	CONST robtarget Target_3690:=[[1119.7,-188.1,-317.9],[-0.081770019911019,-0.37959293775452,0.909310655383545,0.149589429628541],[-1,0,0,1],[9E+09,9E+09,9E+09,9E+09,9E+09,9E+09]];
	CONST robtarget Target_3700:=[[1124.4,-187.9,-319.1],[-0.0822084087134797,-0.376924329069528,0.910420076965927,0.149348957644967],[-1,0,0,1],[9E+09,9E+09,9E+09,9E+09,9E+09,9E+09]];
	CONST robtarget Target_3710:=[[1129.1,-187.6,-320.4],[-0.082652076021253,-0.374348316571166,0.911487931806646,0.14906952197064],[-1,0,0,1],[9E+09,9E+09,9E+09,9E+09,9E+09,9E+09]];
	CONST robtarget Target_3720:=[[1133.8,-187.2,-321.6],[-0.0830604381900551,-0.371848073764742,0.912510779106895,0.148842371853092],[-1,0,0,1],[9E+09,9E+09,9E+09,9E+09,9E+09,9E+09]];
	CONST robtarget Target_3730:=[[1138.6,-187,-322.9],[-0.0834905201851688,-0.369207677745856,0.913582291116862,0.148601551440044],[-1,0,0,1],[9E+09,9E+09,9E+09,9E+09,9E+09,9E+09]];
	CONST robtarget Target_3740:=[[1143.3,-186.7,-324.1],[-0.0839164170034894,-0.366716795237724,0.914590588848913,0.148326942383598],[-1,0,0,1],[9E+09,9E+09,9E+09,9E+09,9E+09,9E+09]];
	CONST robtarget Target_3750:=[[1148,-186.4,-325.4],[-0.0843167371331287,-0.364245178298671,0.915577742852347,0.14809974584311],[-1,0,0,1],[9E+09,9E+09,9E+09,9E+09,9E+09,9E+09]];
	CONST robtarget Target_3760:=[[1152.7,-186.1,-326.6],[-0.0847116064048817,-0.361800877254619,0.916546386353804,0.147874239203031],[-1,0,0,1],[9E+09,9E+09,9E+09,9E+09,9E+09,9E+09]];
	CONST robtarget Target_3770:=[[1157.5,-185.8,-327.9],[-0.0851099118523378,-0.359328899108832,0.917518335176831,0.147645351379778],[-1,0,0,1],[9E+09,9E+09,9E+09,9E+09,9E+09,9E+09]];
	CONST robtarget Target_3780:=[[1157.5,-180.9,-326.9],[-0.085634841189232,-0.362538132200784,0.916590329863401,0.145240985523245],[-1,0,0,1],[9E+09,9E+09,9E+09,9E+09,9E+09,9E+09]];
	CONST robtarget Target_3790:=[[1157.5,-176,-325.8],[-0.0861677390911265,-0.365697677609429,0.915653113093589,0.142897536063477],[-1,0,0,1],[9E+09,9E+09,9E+09,9E+09,9E+09,9E+09]];
	CONST robtarget Target_3800:=[[1157.5,-171.1,-324.9],[-0.0867279055318608,-0.368816467199481,0.914709329423617,0.140568583225226],[-1,0,0,1],[9E+09,9E+09,9E+09,9E+09,9E+09,9E+09]];
	CONST robtarget Target_3810:=[[1157.5,-166.2,-323.9],[-0.0873065476042629,-0.371898546178329,0.913760797007033,0.138239805949448],[-1,0,0,1],[9E+09,9E+09,9E+09,9E+09,9E+09,9E+09]];
	CONST robtarget Target_3820:=[[1157.5,-161.3,-323],[-0.087923551535875,-0.374952346833089,0.912809279452066,0.135865396756779],[-1,0,0,1],[9E+09,9E+09,9E+09,9E+09,9E+09,9E+09]];
	CONST robtarget Target_3830:=[[1157.5,-156.5,-322.1],[-0.0885457305098963,-0.377910274200135,0.911873087948939,0.133532579309003],[-1,0,0,1],[9E+09,9E+09,9E+09,9E+09,9E+09,9E+09]];
	CONST robtarget Target_3840:=[[1157.5,-151.6,-321.2],[-0.0891774776768113,-0.380884851594658,0.910911188916038,0.131205614241488],[-1,0,0,1],[9E+09,9E+09,9E+09,9E+09,9E+09,9E+09]];
	CONST robtarget Target_3850:=[[1157.5,-146.7,-320.4],[-0.0898350121694737,-0.383820989667297,0.909943857926704,0.128892567282967],[-1,0,0,1],[9E+09,9E+09,9E+09,9E+09,9E+09,9E+09]];
	CONST robtarget Target_3860:=[[1157.5,-141.8,-319.6],[-0.090538948270863,-0.386727190520538,0.908972312148108,0.126546887382584],[-1,0,0,1],[9E+09,9E+09,9E+09,9E+09,9E+09,9E+09]];
	CONST robtarget Target_3870:=[[1157.5,-136.9,-318.8],[-0.0912298198832608,-0.389593997110689,0.907997372118494,0.124235299352858],[-1,0,0,1],[9E+09,9E+09,9E+09,9E+09,9E+09,9E+09]];
	CONST robtarget Target_3880:=[[1157.5,-132,-318.1],[-0.091945722049869,-0.392423813800334,0.907017578768495,0.121937059026639],[-1,0,0,1],[9E+09,9E+09,9E+09,9E+09,9E+09,9E+09]];
	CONST robtarget Target_3890:=[[1157.5,-127.1,-317.4],[-0.09267744685106,-0.395219958040731,0.906034447792381,0.119639688335463],[-1,0,0,1],[9E+09,9E+09,9E+09,9E+09,9E+09,9E+09]];
	CONST robtarget Target_3900:=[[1157.5,-122.2,-316.7],[-0.0934459398585867,-0.397990450533941,0.90504850520611,0.117297318093474],[-1,0,0,1],[9E+09,9E+09,9E+09,9E+09,9E+09,9E+09]];
	CONST robtarget Target_3910:=[[1157.5,-117.3,-316],[-0.0942176050684812,-0.400717638074019,0.904057659766507,0.115013761129028],[-1,0,0,1],[9E+09,9E+09,9E+09,9E+09,9E+09,9E+09]];
	CONST robtarget Target_3920:=[[1157.5,-112.4,-315.4],[-0.0950042127207623,-0.403412314824983,0.903063888470925,0.112731172053829],[-1,0,0,1],[9E+09,9E+09,9E+09,9E+09,9E+09,9E+09]];
	CONST robtarget Target_3930:=[[1157.5,-107.6,-314.7],[-0.0958203709921909,-0.406026876380138,0.902086535754033,0.11045593769099],[-1,0,0,1],[9E+09,9E+09,9E+09,9E+09,9E+09,9E+09]];
	CONST robtarget Target_3940:=[[1157.5,-102.7,-314.2],[-0.0966575256864694,-0.408665629753412,0.901086967457954,0.108129565169957],[-1,0,0,1],[9E+09,9E+09,9E+09,9E+09,9E+09,9E+09]];
	CONST robtarget Target_3950:=[[1157.5,-97.8,-313.6],[-0.0974965183603951,-0.411263091531744,0.900083594760464,0.10586132860698],[-1,0,0,1],[9E+09,9E+09,9E+09,9E+09,9E+09,9E+09]];
	CONST robtarget Target_3960:=[[1157.5,-92.9,-313.1],[-0.0983493052491232,-0.413829493044003,0.899077740529287,0.103594311275819],[-1,0,0,1],[9E+09,9E+09,9E+09,9E+09,9E+09,9E+09]];
	CONST robtarget Target_3970:=[[1157.5,-88,-312.6],[-0.0992252665873052,-0.416363081924884,0.898068247921142,0.101338800844204],[-1,0,0,1],[9E+09,9E+09,9E+09,9E+09,9E+09,9E+09]];
	CONST robtarget Target_3980:=[[1157.5,-83.1,-312.1],[-0.100136755641848,-0.418873626645508,0.897055691069865,0.0990383874542113],[-1,0,0,1],[9E+09,9E+09,9E+09,9E+09,9E+09,9E+09]];
	CONST robtarget Target_3990:=[[1157.5,-78.2,-311.6],[-0.101039180167052,-0.421346926627475,0.896041552749548,0.0967852635421828],[-1,0,0,1],[9E+09,9E+09,9E+09,9E+09,9E+09,9E+09]];
	CONST robtarget Target_4000:=[[1157.5,-73.3,-311.2],[-0.101954320538193,-0.423790577515119,0.89502528752291,0.0945335793648495],[-1,0,0,1],[9E+09,9E+09,9E+09,9E+09,9E+09,9E+09]];
	CONST robtarget Target_4010:=[[1157.5,-68.5,-310.8],[-0.102896186994666,-0.42616193510684,0.894025342835322,0.0922879522805532],[-1,0,0,1],[9E+09,9E+09,9E+09,9E+09,9E+09,9E+09]];
	CONST robtarget Target_4020:=[[1157.5,-63.6,-310.5],[-0.103868543102495,-0.428553079264927,0.893002320186698,0.090002445230613],[-1,0,0,1],[9E+09,9E+09,9E+09,9E+09,9E+09,9E+09]];
	CONST robtarget Target_4030:=[[1157.5,-58.7,-310.1],[-0.104830406221372,-0.430908588307866,0.891978581406433,0.0877643707101632],[-1,0,0,1],[9E+09,9E+09,9E+09,9E+09,9E+09,9E+09]];
	CONST robtarget Target_4040:=[[1157.5,-53.8,-309.8],[-0.105814334622865,-0.433234255109494,0.890951696495378,0.0855364325889902],[-1,0,0,1],[9E+09,9E+09,9E+09,9E+09,9E+09,9E+09]];
	CONST robtarget Target_4050:=[[1157.5,-48.9,-309.5],[-0.106809880606017,-0.435532061690535,0.889922999304026,0.0833098310780098],[-1,0,0,1],[9E+09,9E+09,9E+09,9E+09,9E+09,9E+09]];
	CONST robtarget Target_4060:=[[1157.5,-44,-309.3],[-0.107839723601408,-0.437809013192539,0.888890636361769,0.0810388707307653],[-1,0,0,1],[9E+09,9E+09,9E+09,9E+09,9E+09,9E+09]];
	CONST robtarget Target_4070:=[[1157.5,-39.1,-309.1],[-0.10886840289795,-0.4400505689674,0.887857005220818,0.0788232572419922],[-1,0,0,1],[9E+09,9E+09,9E+09,9E+09,9E+09,9E+09]];
	CONST robtarget Target_4080:=[[1157.5,-34.2,-308.8],[-0.109897288481995,-0.442266525786448,0.886823054715504,0.0766014084606349],[-1,0,0,1],[9E+09,9E+09,9E+09,9E+09,9E+09,9E+09]];
	CONST robtarget Target_4090:=[[1157.5,-29.3,-308.7],[-0.110947538224501,-0.444454570827599,0.885786132357125,0.0743888832836221],[-1,0,0,1],[9E+09,9E+09,9E+09,9E+09,9E+09,9E+09]];
	CONST robtarget Target_4100:=[[1157.5,-24.4,-308.5],[-0.112042503144085,-0.44662162946331,0.884743749945618,0.0721394102894673],[-1,0,0,1],[9E+09,9E+09,9E+09,9E+09,9E+09,9E+09]];
	CONST robtarget Target_4110:=[[1157.5,-19.6,-308.4],[-0.113116403345818,-0.448720948594571,0.883722022425974,0.0699255079769918],[-1,0,0,1],[9E+09,9E+09,9E+09,9E+09,9E+09,9E+09]];
	CONST robtarget Target_4120:=[[1157.5,-14.7,-308.3],[-0.114208395342144,-0.450830345502874,0.88267875116301,0.0677249160386389],[-1,0,0,1],[9E+09,9E+09,9E+09,9E+09,9E+09,9E+09]];
	CONST robtarget Target_4130:=[[1157.5,-9.8,-308.2],[-0.115321553262797,-0.452913443093735,0.881632492180146,0.0655324434937342],[-1,0,0,1],[9E+09,9E+09,9E+09,9E+09,9E+09,9E+09]];
	CONST robtarget Target_4140:=[[1157.5,-4.9,-308.2],[-0.116456698651549,-0.454978592783004,0.880583191851778,0.0632894910432632],[-1,0,0,1],[9E+09,9E+09,9E+09,9E+09,9E+09,9E+09]];
	CONST robtarget Target_4150:=[[1157.5,0,-308.2],[-0.117589182842313,-0.457011856882657,0.879533807175913,0.0611001536969137],[-1,0,0,1],[9E+09,9E+09,9E+09,9E+09,9E+09,9E+09]];
	CONST robtarget Target_4160:=[[1162.1,0,-309.4],[-0.117745867154259,-0.454749290253077,0.880705761483944,0.060797660081628],[-1,0,0,1],[9E+09,9E+09,9E+09,9E+09,9E+09,9E+09]];
	CONST robtarget Target_4170:=[[1166.9,0,-310.7],[-0.117907332442503,-0.452402670081197,0.881913476141562,0.0604839289365585],[-1,0,0,1],[9E+09,9E+09,9E+09,9E+09,9E+09,9E+09]];
	CONST robtarget Target_4180:=[[1171.6,0,-312],[-0.118063445251058,-0.450119126040763,0.883081155765986,0.0601786307484635],[-1,0,0,1],[9E+09,9E+09,9E+09,9E+09,9E+09,9E+09]];
	CONST robtarget Target_4190:=[[1176.3,0,-313.3],[-0.118217611912367,-0.447849634992371,0.884234278759815,0.0598752113737095],[-1,0,0,1],[9E+09,9E+09,9E+09,9E+09,9E+09,9E+09]];
	CONST robtarget Target_4200:=[[1181,0,-314.6],[-0.118369853812015,-0.445594206840969,0.885373005081168,0.0595736721365373],[-1,0,0,1],[9E+09,9E+09,9E+09,9E+09,9E+09,9E+09]];
	CONST robtarget Target_4210:=[[1185.7,0,-315.9],[-0.118520192321856,-0.443352847504531,0.88649749458547,0.05927401382815],[-1,0,0,1],[9E+09,9E+09,9E+09,9E+09,9E+09,9E+09]];
	CONST robtarget Target_4220:=[[1190.4,0,-317.1],[-0.118668648788962,-0.441125559029803,0.887607906942775,0.0589762367221873],[-1,0,0,1],[9E+09,9E+09,9E+09,9E+09,9E+09,9E+09]];
	CONST robtarget Target_4230:=[[1195.1,0,-318.4],[-0.118815244525036,-0.438912339707008,0.888704401558589,0.0586803405900602],[-1,0,0,1],[9E+09,9E+09,9E+09,9E+09,9E+09,9E+09]];
	CONST robtarget Target_4240:=[[1199.9,0,-319.7],[-0.118963060887192,-0.436666546379707,0.88981002611204,0.0583800894797157],[-1,0,0,1],[9E+09,9E+09,9E+09,9E+09,9E+09,9E+09]];
	CONST robtarget Target_4250:=[[1204.6,0,-321],[-0.119105960448384,-0.434481744690965,0.890878874385842,0.0580879926402815],[-1,0,0,1],[9E+09,9E+09,9E+09,9E+09,9E+09,9E+09]];
	CONST robtarget Target_4260:=[[1209.3,0,-322.3],[-0.119247063351551,-0.432310985317017,0.891934284166115,0.0577977731866946],[-1,0,0,1],[9E+09,9E+09,9E+09,9E+09,9E+09,9E+09]];
	CONST robtarget Target_4270:=[[1214,0,-323.6],[-0.119386390668427,-0.430154252575755,0.892976413063461,0.0575094290223371],[-1,0,0,1],[9E+09,9E+09,9E+09,9E+09,9E+09,9E+09]];
	CONST robtarget Target_4280:=[[1218.7,0,-324.9],[-0.119523963388954,-0.428011527585619,0.894005418076711,0.0572229576228409],[-1,0,0,1],[9E+09,9E+09,9E+09,9E+09,9E+09,9E+09]];
	CONST robtarget Target_4290:=[[1223.4,0,-326.1],[-0.119659802413315,-0.425882788372245,0.895021455533314,0.0569383560503457],[-1,0,0,1],[9E+09,9E+09,9E+09,9E+09,9E+09,9E+09]];
	CONST robtarget Target_4300:=[[1228.2,0,-327.4],[-0.119796763833562,-0.423723166168958,0.896045888193481,0.0566496255796569],[-1,0,0,1],[9E+09,9E+09,9E+09,9E+09,9E+09,9E+09]];
	CONST robtarget Target_4310:=[[1232.9,0,-328.7],[-0.11992916198956,-0.421622616861546,0.897036188928581,0.0563687928537703],[-1,0,0,1],[9E+09,9E+09,9E+09,9E+09,9E+09,9E+09]];
	CONST robtarget Target_4320:=[[1237.6,0,-330],[-0.120059888974377,-0.419535969212277,0.89801398977622,0.0560898187086545],[-1,0,0,1],[9E+09,9E+09,9E+09,9E+09,9E+09,9E+09]];
	CONST robtarget Target_4330:=[[1242.3,0,-331.3],[-0.120188965254726,-0.417463189853717,0.898979443821632,0.0558126986832536],[-1,0,0,1],[9E+09,9E+09,9E+09,9E+09,9E+09,9E+09]];
	CONST robtarget Target_4340:=[[1247,0,-332.6],[-0.120316411173384,-0.415404242836297,0.89993270322302,0.0555374279712939],[-1,0,0,1],[9E+09,9E+09,9E+09,9E+09,9E+09,9E+09]];
	CONST robtarget Target_4350:=[[1251.8,0,-333.9],[-0.120444906953813,-0.413315725400007,0.900893815293321,0.0552582038451925],[-1,0,0,1],[9E+09,9E+09,9E+09,9E+09,9E+09,9E+09]];
	CONST robtarget Target_4360:=[[1251.8,-5,-333.9],[-0.119365190355739,-0.411088748585182,0.901907684450129,0.0576239607091761],[-1,0,0,1],[9E+09,9E+09,9E+09,9E+09,9E+09,9E+09]];
	CONST robtarget Target_4370:=[[1251.8,-10,-333.9],[-0.118307741993707,-0.408836865218115,0.902915288829416,0.0599973084485274],[-1,0,0,1],[9E+09,9E+09,9E+09,9E+09,9E+09,9E+09]];
	CONST robtarget Target_4380:=[[1251.8,-15,-334],[-0.117260990851089,-0.406560628716403,0.903918121285456,0.0623726319319307],[-1,0,0,1],[9E+09,9E+09,9E+09,9E+09,9E+09,9E+09]];
	CONST robtarget Target_4390:=[[1251.8,-20,-334.1],[-0.116225198631262,-0.404259867017925,0.904916092191274,0.0647497429728289],[-1,0,0,1],[9E+09,9E+09,9E+09,9E+09,9E+09,9E+09]];
	CONST robtarget Target_4400:=[[1251.8,-25,-334.2],[-0.115200628095068,-0.401934408304075,0.905909111119453,0.0671284522279307],[-1,0,0,1],[9E+09,9E+09,9E+09,9E+09,9E+09,9E+09]];
	CONST robtarget Target_4410:=[[1251.8,-30,-334.4],[-0.114177826229758,-0.399576296492031,0.906897618349547,0.0695623253714255],[-1,0,0,1],[9E+09,9E+09,9E+09,9E+09,9E+09,9E+09]];
	CONST robtarget Target_4420:=[[1251.8,-35,-334.6],[-0.113208396368411,-0.397206277971363,0.907877096868025,0.0719041634004291],[-1,0,0,1],[9E+09,9E+09,9E+09,9E+09,9E+09,9E+09]];
	CONST robtarget Target_4430:=[[1251.8,-40,-334.8],[-0.112240868163906,-0.394802969552821,0.90885194146769,0.0743017579637067],[-1,0,0,1],[9E+09,9E+09,9E+09,9E+09,9E+09,9E+09]];
	CONST robtarget Target_4440:=[[1251.8,-45,-335],[-0.111253696234398,-0.392368519801423,0.909824411361592,0.0767404732429802],[-1,0,0,1],[9E+09,9E+09,9E+09,9E+09,9E+09,9E+09]];
	CONST robtarget Target_4450:=[[1251.8,-50,-335.3],[-0.110310416782409,-0.389913691291365,0.910788442329569,0.0791412573296013],[-1,0,0,1],[9E+09,9E+09,9E+09,9E+09,9E+09,9E+09]];
	CONST robtarget Target_4460:=[[1251.8,-55,-335.6],[-0.109390290202297,-0.38743131692568,0.911745622822499,0.0815515685851842],[-1,0,0,1],[9E+09,9E+09,9E+09,9E+09,9E+09,9E+09]];
	CONST robtarget Target_4470:=[[1251.8,-60,-336],[-0.108482698248023,-0.384922590330042,0.912697222791255,0.0839635822459261],[-1,0,0,1],[9E+09,9E+09,9E+09,9E+09,9E+09,9E+09]];
	CONST robtarget Target_4480:=[[1251.8,-65,-336.3],[-0.10758792134765,-0.382387338002196,0.913643125034888,0.086377097613721],[-1,0,0,1],[9E+09,9E+09,9E+09,9E+09,9E+09,9E+09]];
	CONST robtarget Target_4490:=[[1251.8,-70,-336.7],[-0.106706240839152,-0.379825387564897,0.914583210758717,0.0887919125001225],[-1,0,0,1],[9E+09,9E+09,9E+09,9E+09,9E+09,9E+09]];
	CONST robtarget Target_4500:=[[1251.8,-75,-337.1],[-0.105848296774295,-0.377234732453949,0.91551601122939,0.0912169276121816],[-1,0,0,1],[9E+09,9E+09,9E+09,9E+09,9E+09,9E+09]];
	CONST robtarget Target_4510:=[[1251.8,-80,-337.6],[-0.105003845112194,-0.374616877120583,0.91644275072051,0.0936433261898658],[-1,0,0,1],[9E+09,9E+09,9E+09,9E+09,9E+09,9E+09]];
	CONST robtarget Target_4520:=[[1251.8,-85,-338.1],[-0.104173173517156,-0.371971651231437,0.917363299170589,0.0960709005598221],[-1,0,0,1],[9E+09,9E+09,9E+09,9E+09,9E+09,9E+09]];
	CONST robtarget Target_4530:=[[1251.8,-90,-338.6],[-0.103366683650324,-0.369296805579684,0.91827616664258,0.0985092882726507],[-1,0,0,1],[9E+09,9E+09,9E+09,9E+09,9E+09,9E+09]];
	CONST robtarget Target_4540:=[[1251.8,-94.9,-339.1],[-0.102569367780589,-0.366639855644028,0.919164307545986,0.10095403300475],[-1,0,0,1],[9E+09,9E+09,9E+09,9E+09,9E+09,9E+09]];
	CONST robtarget Target_4550:=[[1251.8,-99.9,-339.7],[-0.101791401265309,-0.363909591209621,0.920064048057718,0.103394717107482],[-1,0,0,1],[9E+09,9E+09,9E+09,9E+09,9E+09,9E+09]];
	CONST robtarget Target_4560:=[[1251.8,-105,-340.3],[-0.101043481429939,-0.361102035827114,0.920973980379984,0.105841683873036],[-1,0,0,1],[9E+09,9E+09,9E+09,9E+09,9E+09,9E+09]];
	CONST robtarget Target_4570:=[[1251.8,-110,-340.9],[-0.100305303113894,-0.358312203741803,0.921858683650493,0.108294866891757],[-1,0,0,1],[9E+09,9E+09,9E+09,9E+09,9E+09,9E+09]];
	CONST robtarget Target_4580:=[[1251.8,-114.9,-341.6],[-0.099586379320185,-0.355538933266474,0.922716476741266,0.110765172937249],[-1,0,0,1],[9E+09,9E+09,9E+09,9E+09,9E+09,9E+09]];
	CONST robtarget Target_4590:=[[1251.8,-119.9,-342.3],[-0.0988787294896709,-0.35269196810532,0.923586796329145,0.113220148979633],[-1,0,0,1],[9E+09,9E+09,9E+09,9E+09,9E+09,9E+09]];
	CONST robtarget Target_4600:=[[1251.8,-124.9,-343],[-0.0981776698665501,-0.349805589833328,0.92444729188497,0.115734173809971],[-1,0,0,1],[9E+09,9E+09,9E+09,9E+09,9E+09,9E+09]];
	CONST robtarget Target_4610:=[[1251.8,-129.9,-343.7],[-0.0975211682067817,-0.346894770108699,0.925299498644537,0.118213696461056],[-1,0,0,1],[9E+09,9E+09,9E+09,9E+09,9E+09,9E+09]];
	CONST robtarget Target_4620:=[[1251.8,-134.9,-344.5],[-0.0968808681244795,-0.34395427980659,0.926143868579232,0.120694181662876],[-1,0,0,1],[9E+09,9E+09,9E+09,9E+09,9E+09,9E+09]];
	CONST robtarget Target_4630:=[[1251.8,-139.9,-345.3],[-0.0962570810498641,-0.34098396955735,0.926980220358796,0.123175394930279],[-1,0,0,1],[9E+09,9E+09,9E+09,9E+09,9E+09,9E+09]];
	CONST robtarget Target_4640:=[[1251.8,-144.9,-346.2],[-0.0956501185125098,-0.337983693851527,0.927808369679983,0.125657099563821],[-1,0,0,1],[9E+09,9E+09,9E+09,9E+09,9E+09,9E+09]];
	CONST robtarget Target_4650:=[[1251.8,-149.9,-347],[-0.0950696189951441,-0.334950171594067,0.928626534887739,0.128151897354718],[-1,0,0,1],[9E+09,9E+09,9E+09,9E+09,9E+09,9E+09]];
	CONST robtarget Target_4660:=[[1251.8,-154.9,-347.9],[-0.0945064640355247,-0.331886219394539,0.929436051575064,0.130647203047202],[-1,0,0,1],[9E+09,9E+09,9E+09,9E+09,9E+09,9E+09]];
	CONST robtarget Target_4670:=[[1251.8,-159.9,-348.9],[-0.0939609701945678,-0.328791703294963,0.930236719612129,0.13314277077543],[-1,0,0,1],[9E+09,9E+09,9E+09,9E+09,9E+09,9E+09]];
	CONST robtarget Target_4680:=[[1251.8,-164.9,-349.8],[-0.093442636575496,-0.325663071896759,0.931026631224141,0.13565194146791],[-1,0,0,1],[9E+09,9E+09,9E+09,9E+09,9E+09,9E+09]];
	CONST robtarget Target_4690:=[[1251.8,-169.9,-350.8],[-0.0929425081399444,-0.32250343302878,0.931807201758761,0.138161371648576],[-1,0,0,1],[9E+09,9E+09,9E+09,9E+09,9E+09,9E+09]];
	CONST robtarget Target_4700:=[[1251.8,-174.9,-351.8],[-0.0924700063181994,-0.319309051540198,0.932576424639331,0.14068489521954],[-1,0,0,1],[9E+09,9E+09,9E+09,9E+09,9E+09,9E+09]];
	CONST robtarget Target_4710:=[[1251.8,-179.9,-352.9],[-0.0920162744058036,-0.316083234550579,0.93333577734982,0.143208661746861],[-1,0,0,1],[9E+09,9E+09,9E+09,9E+09,9E+09,9E+09]];
	CONST robtarget Target_4720:=[[1256.5,-179.6,-354.1],[-0.0923098109082863,-0.314168238786619,0.933982120911778,0.143019629299364],[-1,0,0,1],[9E+09,9E+09,9E+09,9E+09,9E+09,9E+09]];
	CONST robtarget Target_4730:=[[1261.2,-179.3,-355.4],[-0.0925904678703637,-0.312277676377353,0.934619019776767,0.142817876918206],[-1,0,0,1],[9E+09,9E+09,9E+09,9E+09,9E+09,9E+09]];
	CONST robtarget Target_4740:=[[1265.9,-179,-356.6],[-0.0928936110909796,-0.310412043924145,0.935245758507429,0.142585101603138],[-1,0,0,1],[9E+09,9E+09,9E+09,9E+09,9E+09,9E+09]];
	CONST robtarget Target_4750:=[[1270.6,-178.7,-357.9],[-0.0931759327644159,-0.30855843130627,0.935858942517041,0.142400771536465],[-1,0,0,1],[9E+09,9E+09,9E+09,9E+09,9E+09,9E+09]];
	CONST robtarget Target_4760:=[[1275.3,-178.5,-359.1],[-0.093462914735115,-0.306670511029906,0.936479291540372,0.142212579436265],[-1,0,0,1],[9E+09,9E+09,9E+09,9E+09,9E+09,9E+09]];
	CONST robtarget Target_4770:=[[1280.1,-178.2,-360.4],[-0.093744445755668,-0.304814801264779,0.937084949590598,0.142027156102845],[-1,0,0,1],[9E+09,9E+09,9E+09,9E+09,9E+09,9E+09]];
	CONST robtarget Target_4780:=[[1284.8,-177.9,-361.6],[-0.0940328166867494,-0.303028934052148,0.937669415667226,0.141800428192085],[-1,0,0,1],[9E+09,9E+09,9E+09,9E+09,9E+09,9E+09]];
	CONST robtarget Target_4790:=[[1289.5,-177.6,-362.9],[-0.0943009704151953,-0.301254085156141,0.9382411439109,0.141622240584786],[-1,0,0,1],[9E+09,9E+09,9E+09,9E+09,9E+09,9E+09]];
	CONST robtarget Target_4800:=[[1294.2,-177.3,-364.1],[-0.0945657720752437,-0.299498165067407,0.938803130092648,0.141445561264098],[-1,0,0,1],[9E+09,9E+09,9E+09,9E+09,9E+09,9E+09]];
	CONST robtarget Target_4810:=[[1298.9,-177,-365.4],[-0.0948437319418863,-0.297769065402197,0.93935842433775,0.141223230477625],[-1,0,0,1],[9E+09,9E+09,9E+09,9E+09,9E+09,9E+09]];
	CONST robtarget Target_4820:=[[1303.6,-176.7,-366.6],[-0.095101903278891,-0.296050262980581,0.939901541372248,0.141049503040362],[-1,0,0,1],[9E+09,9E+09,9E+09,9E+09,9E+09,9E+09]];
	CONST robtarget Target_4830:=[[1308.4,-176.4,-367.9],[-0.0953627832009456,-0.294310263687166,0.940447837135686,0.140873254719873],[-1,0,0,1],[9E+09,9E+09,9E+09,9E+09,9E+09,9E+09]];
	CONST robtarget Target_4840:=[[1313.1,-176.1,-369.1],[-0.0956307502487764,-0.292636132351492,0.940975532659406,0.140655254383064],[-1,0,0,1],[9E+09,9E+09,9E+09,9E+09,9E+09,9E+09]];
	CONST robtarget Target_4850:=[[1317.8,-175.8,-370.4],[-0.0958793438743495,-0.290971597327278,0.94149157647326,0.140485915297344],[-1,0,0,1],[9E+09,9E+09,9E+09,9E+09,9E+09,9E+09]];
	CONST robtarget Target_4860:=[[1322.5,-175.5,-371.6],[-0.0961248966858667,-0.289324553382083,0.94199902432622,0.140318014580593],[-1,0,0,1],[9E+09,9E+09,9E+09,9E+09,9E+09,9E+09]];
	CONST robtarget Target_4870:=[[1327.2,-175.2,-372.9],[-0.0963674569829716,-0.287694771600429,0.942498051677068,0.14015154017471],[-1,0,0,1],[9E+09,9E+09,9E+09,9E+09,9E+09,9E+09]];
	CONST robtarget Target_4880:=[[1331.9,-174.9,-374.1],[-0.0966229425870327,-0.286090126554094,0.942991774856666,0.139939126075453],[-1,0,0,1],[9E+09,9E+09,9E+09,9E+09,9E+09,9E+09]];
	CONST robtarget Target_4890:=[[1336.6,-174.7,-375.4],[-0.0968578276534226,-0.284445199731954,0.943492310384989,0.139756036778756],[-1,0,0,1],[9E+09,9E+09,9E+09,9E+09,9E+09,9E+09]];
	CONST robtarget Target_4900:=[[1341.4,-174.3,-376.6],[-0.0970892315469886,-0.282881705462646,0.943962262021475,0.139595378546212],[-1,0,0,1],[9E+09,9E+09,9E+09,9E+09,9E+09,9E+09]];
	CONST robtarget Target_4910:=[[1346.2,-174,-377.9],[-0.0973411284080376,-0.281290757965059,0.944442959361686,0.139383322947305],[-1,0,0,1],[9E+09,9E+09,9E+09,9E+09,9E+09,9E+09]];
	CONST robtarget Target_4920:=[[1346.2,-169.1,-376.9],[-0.0977467849583902,-0.284347963494082,0.943866533520709,0.136776345128341],[-1,0,0,1],[9E+09,9E+09,9E+09,9E+09,9E+09,9E+09]];
	CONST robtarget Target_4930:=[[1346.2,-164.1,-375.9],[-0.0981717175777088,-0.287429251994673,0.943260441132584,0.134188222881099],[-1,0,0,1],[9E+09,9E+09,9E+09,9E+09,9E+09,9E+09]];
	CONST robtarget Target_4940:=[[1346.2,-159.1,-374.9],[-0.0986201312562024,-0.29049720785679,0.942646751873657,0.131539131517821],[-1,0,0,1],[9E+09,9E+09,9E+09,9E+09,9E+09,9E+09]];
	CONST robtarget Target_4950:=[[1346.2,-154.2,-373.9],[-0.0991022967164904,-0.293486362708794,0.942034904360776,0.128898132862591],[-1,0,0,1],[9E+09,9E+09,9E+09,9E+09,9E+09,9E+09]];
	CONST robtarget Target_4960:=[[1346.2,-149.2,-373],[-0.0995877392212445,-0.296490765638542,0.941391527592563,0.126322998162697],[-1,0,0,1],[9E+09,9E+09,9E+09,9E+09,9E+09,9E+09]];
	CONST robtarget Target_4970:=[[1346.2,-144.2,-372.1],[-0.100079824243535,-0.299473728300579,0.940738559926951,0.123735511085944],[-1,0,0,1],[9E+09,9E+09,9E+09,9E+09,9E+09,9E+09]];
	CONST robtarget Target_4980:=[[1346.2,-139.2,-371.3],[-0.100614451432535,-0.302436882539796,0.940074583777804,0.121113340212912],[-1,0,0,1],[9E+09,9E+09,9E+09,9E+09,9E+09,9E+09]];
	CONST robtarget Target_4990:=[[1346.2,-134.3,-370.4],[-0.101164721884479,-0.30531589436779,0.939411916526386,0.118546002803365],[-1,0,0,1],[9E+09,9E+09,9E+09,9E+09,9E+09,9E+09]];
	CONST robtarget Target_5000:=[[1346.2,-129.3,-369.6],[-0.101741229705465,-0.308227713901319,0.938724195658188,0.115936547503687],[-1,0,0,1],[9E+09,9E+09,9E+09,9E+09,9E+09,9E+09]];
	CONST robtarget Target_5010:=[[1346.2,-124.3,-368.9],[-0.102333534354082,-0.311115175405601,0.938025610436359,0.113327620395202],[-1,0,0,1],[9E+09,9E+09,9E+09,9E+09,9E+09,9E+09]];
	CONST robtarget Target_5020:=[[1346.2,-119.4,-368.1],[-0.102929976384479,-0.313922963777386,0.937331090227515,0.110761997398073],[-1,0,0,1],[9E+09,9E+09,9E+09,9E+09,9E+09,9E+09]];
	CONST robtarget Target_5030:=[[1346.2,-114.4,-367.4],[-0.103545795090149,-0.316752112936713,0.936608882026912,0.108213536018256],[-1,0,0,1],[9E+09,9E+09,9E+09,9E+09,9E+09,9E+09]];
	CONST robtarget Target_5040:=[[1346.2,-109.4,-366.8],[-0.104193781519889,-0.319564811629595,0.935877558597188,0.10561809681534],[-1,0,0,1],[9E+09,9E+09,9E+09,9E+09,9E+09,9E+09]];
	CONST robtarget Target_5050:=[[1346.2,-104.4,-366.1],[-0.10486691842255,-0.322351107250489,0.93513458236786,0.10303400377851],[-1,0,0,1],[9E+09,9E+09,9E+09,9E+09,9E+09,9E+09]];
	CONST robtarget Target_5060:=[[1346.2,-99.5,-365.5],[-0.105542255477612,-0.325060026733112,0.934397086557438,0.100493263266446],[-1,0,0,1],[9E+09,9E+09,9E+09,9E+09,9E+09,9E+09]];
	CONST robtarget Target_5070:=[[1346.2,-94.5,-364.9],[-0.106226744562703,-0.327791645339836,0.933634083043202,0.097958741136734],[-1,0,0,1],[9E+09,9E+09,9E+09,9E+09,9E+09,9E+09]];
	CONST robtarget Target_5080:=[[1346.2,-89.5,-364.4],[-0.10695344372535,-0.330504885042742,0.93286052701095,0.0953872055520313],[-1,0,0,1],[9E+09,9E+09,9E+09,9E+09,9E+09,9E+09]];
	CONST robtarget Target_5090:=[[1346.2,-84.5,-363.8],[-0.107694267553824,-0.333194547303151,0.932077470682332,0.0928166312140292],[-1,0,0,1],[9E+09,9E+09,9E+09,9E+09,9E+09,9E+09]];
	CONST robtarget Target_5100:=[[1346.2,-79.6,-363.4],[-0.108435328560487,-0.3358089775591,0.931301156355231,0.0902899013295485],[-1,0,0,1],[9E+09,9E+09,9E+09,9E+09,9E+09,9E+09]];
	CONST robtarget Target_5110:=[[1346.2,-74.6,-362.9],[-0.109196024009588,-0.338443041336777,0.93049850140805,0.0877785565419249],[-1,0,0,1],[9E+09,9E+09,9E+09,9E+09,9E+09,9E+09]];
	CONST robtarget Target_5120:=[[1346.2,-69.6,-362.5],[-0.109988175498309,-0.341061122451655,0.929686704942729,0.0852205530098301],[-1,0,0,1],[9E+09,9E+09,9E+09,9E+09,9E+09,9E+09]];
	CONST robtarget Target_5130:=[[1346.2,-64.6,-362.1],[-0.110793593146235,-0.343655996914977,0.928865979832894,0.0826639402109412],[-1,0,0,1],[9E+09,9E+09,9E+09,9E+09,9E+09,9E+09]];
	CONST robtarget Target_5140:=[[1346.2,-59.7,-361.7],[-0.111608303834052,-0.346176237032244,0.928051744458803,0.0801595848071462],[-1,0,0,1],[9E+09,9E+09,9E+09,9E+09,9E+09,9E+09]];
	CONST robtarget Target_5150:=[[1346.2,-54.7,-361.3],[-0.112431893149946,-0.348716905236613,0.9272131626012,0.0776617055182264],[-1,0,0,1],[9E+09,9E+09,9E+09,9E+09,9E+09,9E+09]];
	CONST robtarget Target_5160:=[[1346.2,-49.7,-361],[-0.113286516713369,-0.351241776432659,0.926365331062547,0.0751175946417358],[-1,0,0,1],[9E+09,9E+09,9E+09,9E+09,9E+09,9E+09]];
	CONST robtarget Target_5170:=[[1346.2,-44.8,-360.8],[-0.11414938385658,-0.353693912795253,0.925524784908103,0.0726251109297401],[-1,0,0,1],[9E+09,9E+09,9E+09,9E+09,9E+09,9E+09]];
	CONST robtarget Target_5180:=[[1346.2,-39.8,-360.5],[-0.115039747783415,-0.356172521583853,0.924658949304561,0.0700915028338855],[-1,0,0,1],[9E+09,9E+09,9E+09,9E+09,9E+09,9E+09]];
	CONST robtarget Target_5190:=[[1346.2,-34.8,-360.3],[-0.115953593460507,-0.358627450987297,0.923783473952652,0.067566328995428],[-1,0,0,1],[9E+09,9E+09,9E+09,9E+09,9E+09,9E+09]];
	CONST robtarget Target_5200:=[[1346.2,-29.8,-360.1],[-0.116849103303759,-0.361054468657394,0.922903056228464,0.0650838422636147],[-1,0,0,1],[9E+09,9E+09,9E+09,9E+09,9E+09,9E+09]];
	CONST robtarget Target_5210:=[[1346.2,-24.9,-359.9],[-0.117770337947182,-0.363418002553263,0.922029378329369,0.0626045399117393],[-1,0,0,1],[9E+09,9E+09,9E+09,9E+09,9E+09,9E+09]];
	CONST robtarget Target_5220:=[[1346.2,-19.9,-359.8],[-0.118730850208716,-0.365805765459381,0.921128796637897,0.0600904915091507],[-1,0,0,1],[9E+09,9E+09,9E+09,9E+09,9E+09,9E+09]];
	CONST robtarget Target_5230:=[[1346.2,-14.9,-359.7],[-0.119702880851243,-0.36817161364789,0.920220437906222,0.0575780242757909],[-1,0,0,1],[9E+09,9E+09,9E+09,9E+09,9E+09,9E+09]];
	CONST robtarget Target_5240:=[[1346.2,-10,-359.6],[-0.120669259343577,-0.370470009326083,0.919322472788011,0.0551098273118455],[-1,0,0,1],[9E+09,9E+09,9E+09,9E+09,9E+09,9E+09]];
	CONST robtarget Target_5250:=[[1346.2,-5,-359.6],[-0.121644038467576,-0.372786261246687,0.918401460810124,0.0526487237532504],[-1,0,0,1],[9E+09,9E+09,9E+09,9E+09,9E+09,9E+09]];
	CONST robtarget Target_5260:=[[1346.2,0,-359.6],[-0.122660938461861,-0.37508665518371,0.917469103784856,0.0501471721931065],[-1,0,0,1],[9E+09,9E+09,9E+09,9E+09,9E+09,9E+09]];
	CONST robtarget Target_5270:=[[1247,-180.2,-351.6],[-0.0916945348607215,-0.318055947587207,0.932659898238735,0.14345048169453],[-1,0,0,1],[9E+09,9E+09,9E+09,9E+09,9E+09,9E+09]];
	CONST robtarget Target_5280:=[[1242.3,-180.5,-350.4],[-0.0913931135312284,-0.320013657728264,0.931989984090849,0.143642706813763],[-1,0,0,1],[9E+09,9E+09,9E+09,9E+09,9E+09,9E+09]];
	CONST robtarget Target_5290:=[[1237.6,-180.8,-349.1],[-0.091087744358842,-0.321992909345137,0.931308025257883,0.143836543511497],[-1,0,0,1],[9E+09,9E+09,9E+09,9E+09,9E+09,9E+09]];
	CONST robtarget Target_5300:=[[1232.9,-181.1,-347.9],[-0.0907783627727378,-0.323993976593036,0.930613762368532,0.144032000867925],[-1,0,0,1],[9E+09,9E+09,9E+09,9E+09,9E+09,9E+09]];
	CONST robtarget Target_5310:=[[1228.2,-181.4,-346.6],[-0.0904470279388317,-0.326008912409632,0.929904319457681,0.144275711124456],[-1,0,0,1],[9E+09,9E+09,9E+09,9E+09,9E+09,9E+09]];
	CONST robtarget Target_5320:=[[1223.4,-181.7,-345.4],[-0.090121967225503,-0.328101731588239,0.92916796546446,0.144478983616444],[-1,0,0,1],[9E+09,9E+09,9E+09,9E+09,9E+09,9E+09]];
	CONST robtarget Target_5330:=[[1218.7,-182,-344.1],[-0.0897999545630442,-0.330170396324356,0.928434900091322,0.144679348367038],[-1,0,0,1],[9E+09,9E+09,9E+09,9E+09,9E+09,9E+09]];
	CONST robtarget Target_5340:=[[1214,-182.3,-342.9],[-0.0894554700034203,-0.332253759117089,0.927685869361753,0.144927865593746],[-1,0,0,1],[9E+09,9E+09,9E+09,9E+09,9E+09,9E+09]];
	CONST robtarget Target_5350:=[[1209.3,-182.6,-341.6],[-0.0891247139754168,-0.334368581224392,0.926925716846229,0.145131501397497],[-1,0,0,1],[9E+09,9E+09,9E+09,9E+09,9E+09,9E+09]];
	CONST robtarget Target_5360:=[[1204.6,-182.9,-340.4],[-0.0887895322356481,-0.336506913219425,0.926151569677687,0.145336802993827],[-1,0,0,1],[9E+09,9E+09,9E+09,9E+09,9E+09,9E+09]];
	CONST robtarget Target_5370:=[[1199.9,-183.2,-339.1],[-0.0884498527767347,-0.338669042814087,0.925363124454556,0.145543776517121],[-1,0,0,1],[9E+09,9E+09,9E+09,9E+09,9E+09,9E+09]];
	CONST robtarget Target_5380:=[[1195.1,-183.4,-337.9],[-0.0880702742574934,-0.340952949211184,0.924518519574609,0.145808848085359],[-1,0,0,1],[9E+09,9E+09,9E+09,9E+09,9E+09,9E+09]];
	CONST robtarget Target_5390:=[[1190.4,-183.7,-336.6],[-0.0877211398640291,-0.343164103234253,0.923700062175846,0.146019159731608],[-1,0,0,1],[9E+09,9E+09,9E+09,9E+09,9E+09,9E+09]];
	CONST robtarget Target_5400:=[[1185.7,-184,-335.4],[-0.0873672830921968,-0.34539992640377,0.922866348640203,0.146231156847156],[-1,0,0,1],[9E+09,9E+09,9E+09,9E+09,9E+09,9E+09]];
	CONST robtarget Target_5410:=[[1181,-184.3,-334.1],[-0.0870086276767732,-0.34766071109707,0.922017047874772,0.146444843192153],[-1,0,0,1],[9E+09,9E+09,9E+09,9E+09,9E+09,9E+09]];
	CONST robtarget Target_5420:=[[1176.3,-184.6,-332.9],[-0.0866260223795731,-0.349938460600053,0.921149417827701,0.146706360036797],[-1,0,0,1],[9E+09,9E+09,9E+09,9E+09,9E+09,9E+09]];
	CONST robtarget Target_5430:=[[1171.6,-184.9,-331.6],[-0.0862659090477359,-0.352246251074069,0.920266248704867,0.146938092525744],[-1,0,0,1],[9E+09,9E+09,9E+09,9E+09,9E+09,9E+09]];
	CONST robtarget Target_5440:=[[1166.9,-185.2,-330.4],[-0.0858922351502221,-0.354583671052544,0.919368158097704,0.147156834839008],[-1,0,0,1],[9E+09,9E+09,9E+09,9E+09,9E+09,9E+09]];
	CONST robtarget Target_5450:=[[1162.1,-185.5,-329.1],[-0.0855047583298773,-0.357001363171177,0.91843204244788,0.147382313735012],[-1,0,0,1],[9E+09,9E+09,9E+09,9E+09,9E+09,9E+09]];
	CONST robtarget Target_5460:=[[1058.4,-191.9,-301.6],[-0.0755196426375664,-0.416459958972194,0.893006834393729,0.152959732854318],[-1,0,0,1],[9E+09,9E+09,9E+09,9E+09,9E+09,9E+09]];
	CONST robtarget Target_5470:=[[1053.6,-192.3,-300.4],[-0.0749948386695809,-0.41951882253895,0.89157392359611,0.153217722447156],[-1,0,0,1],[9E+09,9E+09,9E+09,9E+09,9E+09,9E+09]];
	CONST robtarget Target_5480:=[[1048.9,-192.5,-299.1],[-0.0744560047898698,-0.422649013071223,0.890094329524097,0.153480290753246],[-1,0,0,1],[9E+09,9E+09,9E+09,9E+09,9E+09,9E+09]];
	CONST robtarget Target_5490:=[[1044.2,-192.8,-297.9],[-0.0738960968592212,-0.425749832850519,0.888609542185254,0.153784031141213],[-1,0,0,1],[9E+09,9E+09,9E+09,9E+09,9E+09,9E+09]];
	CONST robtarget Target_5500:=[[1039.5,-193.1,-296.6],[-0.0733514213142073,-0.428891789433335,0.887097329266413,0.154044572628362],[-1,0,0,1],[9E+09,9E+09,9E+09,9E+09,9E+09,9E+09]];
	CONST robtarget Target_5510:=[[1034.8,-193.4,-295.4],[-0.0727991731829624,-0.432066562567872,0.885555376103445,0.15430632439711],[-1,0,0,1],[9E+09,9E+09,9E+09,9E+09,9E+09,9E+09]];
	CONST robtarget Target_5520:=[[1030.1,-193.7,-294.1],[-0.0722159183465569,-0.435265792974258,0.883981480942423,0.154613362794727],[-1,0,0,1],[9E+09,9E+09,9E+09,9E+09,9E+09,9E+09]];
	CONST robtarget Target_5530:=[[1025.3,-194,-292.9],[-0.0716353435846854,-0.438579183432016,0.882342262981194,0.154883208795643],[-1,0,0,1],[9E+09,9E+09,9E+09,9E+09,9E+09,9E+09]];
	CONST robtarget Target_5540:=[[1020.6,-194.3,-291.6],[-0.0710595030740004,-0.441853803362528,0.880706980576819,0.155148244721643],[-1,0,0,1],[9E+09,9E+09,9E+09,9E+09,9E+09,9E+09]];
	CONST robtarget Target_5550:=[[1015.9,-194.6,-290.4],[-0.0704757269732864,-0.445161665334504,0.879039624191811,0.155414293824337],[-1,0,0,1],[9E+09,9E+09,9E+09,9E+09,9E+09,9E+09]];
	CONST robtarget Target_5560:=[[1011.2,-194.9,-289.1],[-0.0698599262628231,-0.448494319419836,0.877338099476652,0.155725063356508],[-1,0,0,1],[9E+09,9E+09,9E+09,9E+09,9E+09,9E+09]];
	CONST robtarget Target_5570:=[[1006.5,-195.2,-287.9],[-0.0692598520335908,-0.451868831293863,0.875604850746204,0.155992876603775],[-1,0,0,1],[9E+09,9E+09,9E+09,9E+09,9E+09,9E+09]];
	CONST robtarget Target_5580:=[[1001.8,-195.5,-286.6],[-0.0686583135132066,-0.455272740455241,0.873836494953086,0.156277150831474],[-1,0,0,1],[9E+09,9E+09,9E+09,9E+09,9E+09,9E+09]];
	CONST robtarget Target_5590:=[[997.1,-195.8,-285.4],[-0.0680417113457267,-0.458714001293542,0.87203494948929,0.156546598186054],[-1,0,0,1],[9E+09,9E+09,9E+09,9E+09,9E+09,9E+09]];
	CONST robtarget Target_5600:=[[992.3,-196.1,-284.1],[-0.0674028023794809,-0.462266046873075,0.870157221438666,0.156822747450342],[-1,0,0,1],[9E+09,9E+09,9E+09,9E+09,9E+09,9E+09]];
	CONST robtarget Target_5610:=[[987.6,-196.4,-282.9],[-0.0667443729406992,-0.465766124616528,0.86828286007232,0.157136821735347],[-1,0,0,1],[9E+09,9E+09,9E+09,9E+09,9E+09,9E+09]];
	CONST robtarget Target_5620:=[[982.9,-196.6,-281.6],[-0.0660933755521842,-0.46935615793945,0.866347508185939,0.157411745979934],[-1,0,0,1],[9E+09,9E+09,9E+09,9E+09,9E+09,9E+09]];
	CONST robtarget Target_5630:=[[978.2,-197,-280.4],[-0.0654513013274054,-0.472883025030647,0.864427470973437,0.157679799653864],[-1,0,0,1],[9E+09,9E+09,9E+09,9E+09,9E+09,9E+09]];
	CONST robtarget Target_5640:=[[973.5,-197.2,-279.1],[-0.0647831891782489,-0.476538276592348,0.862417809926292,0.157955469877521],[-1,0,0,1],[9E+09,9E+09,9E+09,9E+09,9E+09,9E+09]];
	CONST robtarget Target_5650:=[[869.7,-203.7,-251.6],[-0.0477830710999151,-0.563979721183965,0.807912615766751,0.164075767541839],[-1,0,0,1],[9E+09,9E+09,9E+09,9E+09,9E+09,9E+09]];
	CONST robtarget Target_5660:=[[865,-204,-250.3],[-0.0468856267688857,-0.568231430194026,0.804921520355919,0.164365829204422],[-1,0,0,1],[9E+09,9E+09,9E+09,9E+09,9E+09,9E+09]];
	CONST robtarget Target_5670:=[[860.2,-204.3,-249.1],[-0.0459901904631258,-0.572604680792359,0.801816370328713,0.16461862041924],[-1,0,0,1],[9E+09,9E+09,9E+09,9E+09,9E+09,9E+09]];
	CONST robtarget Target_5680:=[[855.5,-204.6,-247.9],[-0.0451051805643158,-0.576903849032486,0.798728715624983,0.164863308512928],[-1,0,0,1],[9E+09,9E+09,9E+09,9E+09,9E+09,9E+09]];
	CONST robtarget Target_5690:=[[850.8,-204.9,-246.6],[-0.0442117627725604,-0.58122061137896,0.795592994627718,0.165105141773693],[-1,0,0,1],[9E+09,9E+09,9E+09,9E+09,9E+09,9E+09]];
	CONST robtarget Target_5700:=[[846.1,-205.2,-245.3],[-0.0432792420588702,-0.585545172332437,0.792409080300039,0.165383215058337],[-1,0,0,1],[9E+09,9E+09,9E+09,9E+09,9E+09,9E+09]];
	CONST robtarget Target_5710:=[[841.4,-205.5,-244.1],[-0.042369168495389,-0.589893666567888,0.789177268759606,0.165618701169982],[-1,0,0,1],[9E+09,9E+09,9E+09,9E+09,9E+09,9E+09]];
	CONST robtarget Target_5720:=[[836.7,-205.7,-242.8],[-0.0414460623868268,-0.594280009004696,0.785879488395744,0.165852116443685],[-1,0,0,1],[9E+09,9E+09,9E+09,9E+09,9E+09,9E+09]];
	CONST robtarget Target_5730:=[[832,-206,-241.6],[-0.0405203170220552,-0.598654293350079,0.782552449639827,0.166080716895896],[-1,0,0,1],[9E+09,9E+09,9E+09,9E+09,9E+09,9E+09]];
	CONST robtarget Target_5740:=[[827.3,-206.3,-240.3],[-0.0395868816896496,-0.603040074957237,0.779177750824128,0.166305680643543],[-1,0,0,1],[9E+09,9E+09,9E+09,9E+09,9E+09,9E+09]];
	CONST robtarget Target_5750:=[[822.5,-206.6,-239.1],[-0.0385936457931231,-0.607522308703406,0.775681395048548,0.166569950193959],[-1,0,0,1],[9E+09,9E+09,9E+09,9E+09,9E+09,9E+09]];
	CONST robtarget Target_5760:=[[817.8,-206.9,-237.8],[-0.0376450070876776,-0.611927170340272,0.772211188986617,0.166786903696278],[-1,0,0,1],[9E+09,9E+09,9E+09,9E+09,9E+09,9E+09]];
	CONST robtarget Target_5770:=[[813.1,-207.2,-236.6],[-0.0366892387091784,-0.616339415627857,0.768694156957296,0.166999753191925],[-1,0,0,1],[9E+09,9E+09,9E+09,9E+09,9E+09,9E+09]];
	CONST robtarget Target_5780:=[[808.4,-207.5,-235.4],[-0.0357299876826028,-0.620753454512114,0.765130252072654,0.167225040154622],[-1,0,0,1],[9E+09,9E+09,9E+09,9E+09,9E+09,9E+09]];
	CONST robtarget Target_5790:=[[803.7,-207.8,-234.1],[-0.0347604944167214,-0.625176161610856,0.761520794777794,0.16742925103583],[-1,0,0,1],[9E+09,9E+09,9E+09,9E+09,9E+09,9E+09]];
	CONST robtarget Target_5800:=[[798.9,-208.1,-232.8],[-0.0337304773604137,-0.629688375941923,0.75778715982875,0.167670583285617],[-1,0,0,1],[9E+09,9E+09,9E+09,9E+09,9E+09,9E+09]];
	CONST robtarget Target_5810:=[[794.2,-208.4,-231.6],[-0.0327479318751579,-0.634115576754324,0.75408637815255,0.167865251199289],[-1,0,0,1],[9E+09,9E+09,9E+09,9E+09,9E+09,9E+09]];
	CONST robtarget Target_5820:=[[789.5,-208.7,-230.3],[-0.0317593997810374,-0.63854274253144,0.750341253269555,0.168055080636822],[-1,0,0,1],[9E+09,9E+09,9E+09,9E+09,9E+09,9E+09]];
	CONST robtarget Target_5830:=[[784.8,-209,-229.1],[-0.0307651390229622,-0.642968328984431,0.746552448472756,0.168239935280534],[-1,0,0,1],[9E+09,9E+09,9E+09,9E+09,9E+09,9E+09]];
	CONST robtarget Target_5840:=[[681,-215.4,-201.6],[-0.00778880261753513,-0.737023119823921,0.65382583781393,0.171020551998035],[-1,0,0,1],[9E+09,9E+09,9E+09,9E+09,9E+09,9E+09]];
	CONST robtarget Target_5850:=[[676.3,-215.7,-200.3],[-0.00674962721138414,-0.740981822113494,0.649336002887133,0.171064716363237],[-1,0,0,1],[9E+09,9E+09,9E+09,9E+09,9E+09,9E+09]];
	CONST robtarget Target_5860:=[[671.6,-216,-199.1],[-0.00571266089965787,-0.744903909189969,0.644832901937839,0.171102484369377],[-1,0,0,1],[9E+09,9E+09,9E+09,9E+09,9E+09,9E+09]];
	CONST robtarget Target_5870:=[[666.9,-216.3,-197.8],[-0.00467823838086147,-0.748788327367839,0.640318160093673,0.171133891259386],[-1,0,0,1],[9E+09,9E+09,9E+09,9E+09,9E+09,9E+09]];
	CONST robtarget Target_5880:=[[662.2,-216.6,-196.6],[-0.00360764788769451,-0.7526256103041,0.63579528491276,0.171190044318594],[-1,0,0,1],[9E+09,9E+09,9E+09,9E+09,9E+09,9E+09]];
	CONST robtarget Target_5890:=[[657.4,-216.9,-195.3],[-0.00255755580854608,-0.756511214628875,0.631166963444428,0.171208952176486],[-1,0,0,1],[9E+09,9E+09,9E+09,9E+09,9E+09,9E+09]];
	CONST robtarget Target_5900:=[[652.7,-217.2,-194.1],[-0.00153262884980755,-0.760275915333536,0.626627071045187,0.171221194499667],[-1,0,0,1],[9E+09,9E+09,9E+09,9E+09,9E+09,9E+09]];
	CONST robtarget Target_5910:=[[648,-217.5,-192.8],[-0.000511535880873687,-0.763999243627504,0.62208207604746,0.171227289671146],[-1,0,0,1],[9E+09,9E+09,9E+09,9E+09,9E+09,9E+09]];
	CONST robtarget Target_5920:=[[643.3,-217.8,-191.6],[0.000505419678604915,-0.767680414947257,0.617533589458358,0.171227307833863],[-1,0,0,1],[9E+09,9E+09,9E+09,9E+09,9E+09,9E+09]];
	CONST robtarget Target_5930:=[[638.6,-218.1,-190.3],[0.00155789400513257,-0.77131029461782,0.612985339875262,0.171251205779257],[-1,0,0,1],[9E+09,9E+09,9E+09,9E+09,9E+09,9E+09]];
	CONST robtarget Target_5940:=[[633.9,-218.4,-189.1],[0.00256587096633776,-0.774905033947616,0.608434701383857,0.171239069200825],[-1,0,0,1],[9E+09,9E+09,9E+09,9E+09,9E+09,9E+09]];
	CONST robtarget Target_5950:=[[629.1,-218.7,-187.8],[0.00358974474052876,-0.778529300573558,0.603790299387018,0.171220665362796],[-1,0,0,1],[9E+09,9E+09,9E+09,9E+09,9E+09,9E+09]];
	CONST robtarget Target_5960:=[[624.4,-218.9,-186.6],[0.00458106569260151,-0.782012243707725,0.599272432351621,0.171197010346854],[-1,0,0,1],[9E+09,9E+09,9E+09,9E+09,9E+09,9E+09]];
	CONST robtarget Target_5970:=[[619.7,-219.3,-185.3],[0.00561999404124486,-0.78548535344611,0.594704125190122,0.171196316170846],[-1,0,0,1],[9E+09,9E+09,9E+09,9E+09,9E+09,9E+09]];
	CONST robtarget Target_5980:=[[615,-219.5,-184.1],[0.00659971422524121,-0.788876173727834,0.590198796610973,0.171161347200929],[-1,0,0,1],[9E+09,9E+09,9E+09,9E+09,9E+09,9E+09]];
	CONST robtarget Target_5990:=[[610.3,-219.8,-182.8],[0.00757988026613238,-0.792243418895945,0.5856710699809,0.171120742222102],[-1,0,0,1],[9E+09,9E+09,9E+09,9E+09,9E+09,9E+09]];
	CONST robtarget Target_6000:=[[605.6,-220.1,-181.6],[0.00855378584535725,-0.795564255560035,0.581152090482101,0.171074825007082],[-1,0,0,1],[9E+09,9E+09,9E+09,9E+09,9E+09,9E+09]];
	CONST robtarget Target_6010:=[[600.8,-220.4,-180.3],[0.00954125404368884,-0.798905975122599,0.576549633518153,0.171022593462869],[-1,0,0,1],[9E+09,9E+09,9E+09,9E+09,9E+09,9E+09]];
	CONST robtarget Target_6020:=[[596.1,-220.7,-179.1],[0.0105444478776632,-0.802119716707681,0.572055924579113,0.171011092744536],[-1,0,0,1],[9E+09,9E+09,9E+09,9E+09,9E+09,9E+09]];
    !***********************************************************
    !
    ! Module:  test
    !
    ! Description:
    !   <Insert description>
    !
    ! Author: ModuleWriter
    ! Version: 1.0
    !
    !***********************************************************


    !***********************************************************
    !
    ! Procedure main
    !
    !   This is the entry point of your program
    !
    !***********************************************************
    PROC main()
        Path_10;
      !Add your code here
    ENDPROC
      PROC Path_10()
SetDO drillDone,0;
MoveAbsJ jHome, v100, fine, tool0\WObj:= wobj0;
WaitTime 2;
confL \Off;
confJ \Off;
        MoveJ RelTool(Target_10,0,0,-10),v60,z10,DrillTool\WObj:=FakeWing;
SetDO drillDone,1;
WaitUntil drillDone = 0;
        MoveL Target_10,v30,fine,DrillTool\WObj:=FakeWing;
SetDO drillDone,1;
WaitUntil drillDone = 0;
        MoveL RelTool(Target_10,0,0,-10),v30,z10,DrillTool\WObj:=FakeWing;
        MoveL RelTool(Target_20,0,0,-10),v30,z10,DrillTool\WObj:=FakeWing;
        MoveL Target_20,v30,fine,DrillTool\WObj:=FakeWing;
SetDO drillDone,1;
WaitUntil drillDone = 0;
        MoveL RelTool(Target_20,0,0,-10),v30,z10,DrillTool\WObj:=FakeWing;
        MoveL RelTool(Target_30,0,0,-10),v30,z10,DrillTool\WObj:=FakeWing;
        MoveL Target_30,v30,fine,DrillTool\WObj:=FakeWing;
SetDO drillDone,1;
WaitUntil drillDone = 0;
        MoveL RelTool(Target_30,0,0,-10),v30,z10,DrillTool\WObj:=FakeWing;
        MoveL RelTool(Target_40,0,0,-10),v30,z10,DrillTool\WObj:=FakeWing;
        MoveL Target_40,v30,fine,DrillTool\WObj:=FakeWing;
SetDO drillDone,1;
WaitUntil drillDone = 0;
        MoveL RelTool(Target_40,0,0,-10),v30,z10,DrillTool\WObj:=FakeWing;
        MoveL RelTool(Target_50,0,0,-10),v30,z10,DrillTool\WObj:=FakeWing;
        MoveL Target_50,v30,fine,DrillTool\WObj:=FakeWing;
SetDO drillDone,1;
WaitUntil drillDone = 0;
        MoveL RelTool(Target_50,0,0,-10),v30,z10,DrillTool\WObj:=FakeWing;
        MoveL RelTool(Target_60,0,0,-10),v30,z10,DrillTool\WObj:=FakeWing;
        MoveL Target_60,v30,fine,DrillTool\WObj:=FakeWing;
SetDO drillDone,1;
WaitUntil drillDone = 0;
        MoveL RelTool(Target_60,0,0,-10),v30,z10,DrillTool\WObj:=FakeWing;
        MoveL RelTool(Target_70,0,0,-10),v30,z10,DrillTool\WObj:=FakeWing;
        MoveL Target_70,v30,fine,DrillTool\WObj:=FakeWing;
SetDO drillDone,1;
WaitUntil drillDone = 0;
        MoveL RelTool(Target_70,0,0,-10),v30,z10,DrillTool\WObj:=FakeWing;
        MoveL RelTool(Target_80,0,0,-10),v30,z10,DrillTool\WObj:=FakeWing;
        MoveL Target_80,v30,fine,DrillTool\WObj:=FakeWing;
SetDO drillDone,1;
WaitUntil drillDone = 0;
        MoveL RelTool(Target_80,0,0,-10),v30,z10,DrillTool\WObj:=FakeWing;
        MoveL RelTool(Target_90,0,0,-10),v30,z10,DrillTool\WObj:=FakeWing;
        MoveL Target_90,v30,fine,DrillTool\WObj:=FakeWing;
SetDO drillDone,1;
WaitUntil drillDone = 0;
        MoveL RelTool(Target_90,0,0,-10),v30,z10,DrillTool\WObj:=FakeWing;
        MoveL RelTool(Target_100,0,0,-10),v30,z10,DrillTool\WObj:=FakeWing;
        MoveL Target_100,v30,fine,DrillTool\WObj:=FakeWing;
SetDO drillDone,1;
WaitUntil drillDone = 0;
        MoveL RelTool(Target_100,0,0,-10),v30,z10,DrillTool\WObj:=FakeWing;
        MoveL RelTool(Target_110,0,0,-10),v30,z10,DrillTool\WObj:=FakeWing;
        MoveL Target_110,v30,fine,DrillTool\WObj:=FakeWing;
SetDO drillDone,1;
WaitUntil drillDone = 0;
        MoveL RelTool(Target_110,0,0,-10),v30,z10,DrillTool\WObj:=FakeWing;
        MoveL RelTool(Target_120,0,0,-10),v30,z10,DrillTool\WObj:=FakeWing;
        MoveL Target_120,v30,fine,DrillTool\WObj:=FakeWing;
SetDO drillDone,1;
WaitUntil drillDone = 0;
        MoveL RelTool(Target_120,0,0,-10),v30,z10,DrillTool\WObj:=FakeWing;
        MoveL RelTool(Target_130,0,0,-10),v30,z10,DrillTool\WObj:=FakeWing;
        MoveL Target_130,v30,fine,DrillTool\WObj:=FakeWing;
SetDO drillDone,1;
WaitUntil drillDone = 0;
        MoveL RelTool(Target_130,0,0,-10),v30,z10,DrillTool\WObj:=FakeWing;
        MoveL RelTool(Target_140,0,0,-10),v30,z10,DrillTool\WObj:=FakeWing;
        MoveL Target_140,v30,fine,DrillTool\WObj:=FakeWing;
SetDO drillDone,1;
WaitUntil drillDone = 0;
        MoveL RelTool(Target_140,0,0,-10),v30,z10,DrillTool\WObj:=FakeWing;
        MoveL RelTool(Target_150,0,0,-10),v30,z10,DrillTool\WObj:=FakeWing;
        MoveL Target_150,v30,fine,DrillTool\WObj:=FakeWing;
SetDO drillDone,1;
WaitUntil drillDone = 0;
        MoveL RelTool(Target_150,0,0,-10),v30,z10,DrillTool\WObj:=FakeWing;
        MoveL RelTool(Target_160,0,0,-10),v30,z10,DrillTool\WObj:=FakeWing;
        MoveL Target_160,v30,fine,DrillTool\WObj:=FakeWing;
SetDO drillDone,1;
WaitUntil drillDone = 0;
        MoveL RelTool(Target_160,0,0,-10),v30,z10,DrillTool\WObj:=FakeWing;
        MoveL RelTool(Target_170,0,0,-10),v30,z10,DrillTool\WObj:=FakeWing;
        MoveL Target_170,v30,fine,DrillTool\WObj:=FakeWing;
SetDO drillDone,1;
WaitUntil drillDone = 0;
        MoveL RelTool(Target_170,0,0,-10),v30,z10,DrillTool\WObj:=FakeWing;
        MoveL RelTool(Target_180,0,0,-10),v30,z10,DrillTool\WObj:=FakeWing;
        MoveL Target_180,v30,fine,DrillTool\WObj:=FakeWing;
SetDO drillDone,1;
WaitUntil drillDone = 0;
        MoveL RelTool(Target_180,0,0,-10),v30,z10,DrillTool\WObj:=FakeWing;
        MoveL RelTool(Target_190,0,0,-10),v30,z10,DrillTool\WObj:=FakeWing;
        MoveL Target_190,v30,fine,DrillTool\WObj:=FakeWing;
SetDO drillDone,1;
WaitUntil drillDone = 0;
        MoveL RelTool(Target_190,0,0,-10),v30,z10,DrillTool\WObj:=FakeWing;
        MoveL RelTool(Target_200,0,0,-10),v30,z10,DrillTool\WObj:=FakeWing;
        MoveL Target_200,v30,fine,DrillTool\WObj:=FakeWing;
SetDO drillDone,1;
WaitUntil drillDone = 0;
        MoveL RelTool(Target_200,0,0,-10),v30,z10,DrillTool\WObj:=FakeWing;
        MoveL RelTool(Target_210,0,0,-10),v30,z10,DrillTool\WObj:=FakeWing;
        MoveL Target_210,v30,fine,DrillTool\WObj:=FakeWing;
SetDO drillDone,1;
WaitUntil drillDone = 0;
        MoveL RelTool(Target_210,0,0,-10),v30,z10,DrillTool\WObj:=FakeWing;
        MoveL RelTool(Target_220,0,0,-10),v30,z10,DrillTool\WObj:=FakeWing;
        MoveL Target_220,v30,fine,DrillTool\WObj:=FakeWing;
SetDO drillDone,1;
WaitUntil drillDone = 0;
        MoveL RelTool(Target_220,0,0,-10),v30,z10,DrillTool\WObj:=FakeWing;
        MoveL RelTool(Target_230,0,0,-10),v30,z10,DrillTool\WObj:=FakeWing;
        MoveL Target_230,v30,fine,DrillTool\WObj:=FakeWing;
SetDO drillDone,1;
WaitUntil drillDone = 0;
        MoveL RelTool(Target_230,0,0,-10),v30,z10,DrillTool\WObj:=FakeWing;
        MoveL RelTool(Target_240,0,0,-10),v30,z10,DrillTool\WObj:=FakeWing;
        MoveL Target_240,v30,fine,DrillTool\WObj:=FakeWing;
SetDO drillDone,1;
WaitUntil drillDone = 0;
        MoveL RelTool(Target_240,0,0,-10),v30,z10,DrillTool\WObj:=FakeWing;
        MoveL RelTool(Target_250,0,0,-10),v30,z10,DrillTool\WObj:=FakeWing;
        MoveL Target_250,v30,fine,DrillTool\WObj:=FakeWing;
SetDO drillDone,1;
WaitUntil drillDone = 0;
        MoveL RelTool(Target_250,0,0,-10),v30,z10,DrillTool\WObj:=FakeWing;
        MoveL RelTool(Target_260,0,0,-10),v30,z10,DrillTool\WObj:=FakeWing;
        MoveL Target_260,v30,fine,DrillTool\WObj:=FakeWing;
SetDO drillDone,1;
WaitUntil drillDone = 0;
        MoveL RelTool(Target_260,0,0,-10),v30,z10,DrillTool\WObj:=FakeWing;
        MoveL RelTool(Target_270,0,0,-10),v30,z10,DrillTool\WObj:=FakeWing;
        MoveL Target_270,v30,fine,DrillTool\WObj:=FakeWing;
SetDO drillDone,1;
WaitUntil drillDone = 0;
        MoveL RelTool(Target_270,0,0,-10),v30,z10,DrillTool\WObj:=FakeWing;
        MoveL RelTool(Target_280,0,0,-10),v30,z10,DrillTool\WObj:=FakeWing;
        MoveL Target_280,v30,fine,DrillTool\WObj:=FakeWing;
SetDO drillDone,1;
WaitUntil drillDone = 0;
        MoveL RelTool(Target_280,0,0,-10),v30,z10,DrillTool\WObj:=FakeWing;
        MoveL RelTool(Target_290,0,0,-10),v30,z10,DrillTool\WObj:=FakeWing;
        MoveL Target_290,v30,fine,DrillTool\WObj:=FakeWing;
SetDO drillDone,1;
WaitUntil drillDone = 0;
        MoveL RelTool(Target_290,0,0,-10),v30,z10,DrillTool\WObj:=FakeWing;
        MoveL RelTool(Target_300,0,0,-10),v30,z10,DrillTool\WObj:=FakeWing;
        MoveL Target_300,v30,fine,DrillTool\WObj:=FakeWing;
SetDO drillDone,1;
WaitUntil drillDone = 0;
        MoveL RelTool(Target_300,0,0,-10),v30,z10,DrillTool\WObj:=FakeWing;
        MoveL RelTool(Target_310,0,0,-10),v30,z10,DrillTool\WObj:=FakeWing;
        MoveL Target_310,v30,fine,DrillTool\WObj:=FakeWing;
SetDO drillDone,1;
WaitUntil drillDone = 0;
        MoveL RelTool(Target_310,0,0,-10),v30,z10,DrillTool\WObj:=FakeWing;
        MoveL RelTool(Target_320,0,0,-10),v30,z10,DrillTool\WObj:=FakeWing;
        MoveL Target_320,v30,fine,DrillTool\WObj:=FakeWing;
SetDO drillDone,1;
WaitUntil drillDone = 0;
        MoveL RelTool(Target_320,0,0,-10),v30,z10,DrillTool\WObj:=FakeWing;
        MoveL RelTool(Target_330,0,0,-10),v30,z10,DrillTool\WObj:=FakeWing;
        MoveL Target_330,v30,fine,DrillTool\WObj:=FakeWing;
SetDO drillDone,1;
WaitUntil drillDone = 0;
        MoveL RelTool(Target_330,0,0,-10),v30,z10,DrillTool\WObj:=FakeWing;
        MoveL RelTool(Target_340,0,0,-10),v30,z10,DrillTool\WObj:=FakeWing;
        MoveL Target_340,v30,fine,DrillTool\WObj:=FakeWing;
SetDO drillDone,1;
WaitUntil drillDone = 0;
        MoveL RelTool(Target_340,0,0,-10),v30,z10,DrillTool\WObj:=FakeWing;
        MoveL RelTool(Target_350,0,0,-10),v30,z10,DrillTool\WObj:=FakeWing;
        MoveL Target_350,v30,fine,DrillTool\WObj:=FakeWing;
SetDO drillDone,1;
WaitUntil drillDone = 0;
        MoveL RelTool(Target_350,0,0,-10),v30,z10,DrillTool\WObj:=FakeWing;
        MoveL RelTool(Target_360,0,0,-10),v30,z10,DrillTool\WObj:=FakeWing;
        MoveL Target_360,v30,fine,DrillTool\WObj:=FakeWing;
SetDO drillDone,1;
WaitUntil drillDone = 0;
        MoveL RelTool(Target_360,0,0,-10),v30,z10,DrillTool\WObj:=FakeWing;
        MoveL RelTool(Target_370,0,0,-10),v30,z10,DrillTool\WObj:=FakeWing;
        MoveL Target_370,v30,fine,DrillTool\WObj:=FakeWing;
SetDO drillDone,1;
WaitUntil drillDone = 0;
        MoveL RelTool(Target_370,0,0,-10),v30,z10,DrillTool\WObj:=FakeWing;
        MoveL RelTool(Target_380,0,0,-10),v30,z10,DrillTool\WObj:=FakeWing;
        MoveL Target_380,v30,fine,DrillTool\WObj:=FakeWing;
SetDO drillDone,1;
WaitUntil drillDone = 0;
        MoveL RelTool(Target_380,0,0,-10),v30,z10,DrillTool\WObj:=FakeWing;
        MoveL RelTool(Target_390,0,0,-10),v30,z10,DrillTool\WObj:=FakeWing;
        MoveL Target_390,v30,fine,DrillTool\WObj:=FakeWing;
SetDO drillDone,1;
WaitUntil drillDone = 0;
        MoveL RelTool(Target_390,0,0,-10),v30,z10,DrillTool\WObj:=FakeWing;
        MoveL RelTool(Target_400,0,0,-10),v30,z10,DrillTool\WObj:=FakeWing;
        MoveL Target_400,v30,fine,DrillTool\WObj:=FakeWing;
SetDO drillDone,1;
WaitUntil drillDone = 0;
        MoveL RelTool(Target_400,0,0,-10),v30,z10,DrillTool\WObj:=FakeWing;
        MoveL RelTool(Target_410,0,0,-10),v30,z10,DrillTool\WObj:=FakeWing;
        MoveL Target_410,v30,fine,DrillTool\WObj:=FakeWing;
SetDO drillDone,1;
WaitUntil drillDone = 0;
        MoveL RelTool(Target_410,0,0,-10),v30,z10,DrillTool\WObj:=FakeWing;
        MoveL RelTool(Target_420,0,0,-10),v30,z10,DrillTool\WObj:=FakeWing;
        MoveL Target_420,v30,fine,DrillTool\WObj:=FakeWing;
SetDO drillDone,1;
WaitUntil drillDone = 0;
        MoveL RelTool(Target_420,0,0,-10),v30,z10,DrillTool\WObj:=FakeWing;
        MoveL RelTool(Target_430,0,0,-10),v30,z10,DrillTool\WObj:=FakeWing;
        MoveL Target_430,v30,fine,DrillTool\WObj:=FakeWing;
SetDO drillDone,1;
WaitUntil drillDone = 0;
        MoveL RelTool(Target_430,0,0,-10),v30,z10,DrillTool\WObj:=FakeWing;
        MoveL RelTool(Target_440,0,0,-10),v30,z10,DrillTool\WObj:=FakeWing;
        MoveL Target_440,v30,fine,DrillTool\WObj:=FakeWing;
SetDO drillDone,1;
WaitUntil drillDone = 0;
        MoveL RelTool(Target_440,0,0,-10),v30,z10,DrillTool\WObj:=FakeWing;
        MoveL RelTool(Target_450,0,0,-10),v30,z10,DrillTool\WObj:=FakeWing;
        MoveL Target_450,v30,fine,DrillTool\WObj:=FakeWing;
SetDO drillDone,1;
WaitUntil drillDone = 0;
        MoveL RelTool(Target_450,0,0,-10),v30,z10,DrillTool\WObj:=FakeWing;
        MoveL RelTool(Target_460,0,0,-10),v30,z10,DrillTool\WObj:=FakeWing;
        MoveL Target_460,v30,fine,DrillTool\WObj:=FakeWing;
SetDO drillDone,1;
WaitUntil drillDone = 0;
        MoveL RelTool(Target_460,0,0,-10),v30,z10,DrillTool\WObj:=FakeWing;
        MoveL RelTool(Target_470,0,0,-10),v30,z10,DrillTool\WObj:=FakeWing;
        MoveL Target_470,v30,fine,DrillTool\WObj:=FakeWing;
SetDO drillDone,1;
WaitUntil drillDone = 0;
        MoveL RelTool(Target_470,0,0,-10),v30,z10,DrillTool\WObj:=FakeWing;
        MoveL RelTool(Target_480,0,0,-10),v30,z10,DrillTool\WObj:=FakeWing;
        MoveL Target_480,v30,fine,DrillTool\WObj:=FakeWing;
SetDO drillDone,1;
WaitUntil drillDone = 0;
        MoveL RelTool(Target_480,0,0,-10),v30,z10,DrillTool\WObj:=FakeWing;
        MoveL RelTool(Target_490,0,0,-10),v30,z10,DrillTool\WObj:=FakeWing;
        MoveL Target_490,v30,fine,DrillTool\WObj:=FakeWing;
SetDO drillDone,1;
WaitUntil drillDone = 0;
        MoveL RelTool(Target_490,0,0,-10),v30,z10,DrillTool\WObj:=FakeWing;
        MoveL RelTool(Target_500,0,0,-10),v30,z10,DrillTool\WObj:=FakeWing;
        MoveL Target_500,v30,fine,DrillTool\WObj:=FakeWing;
SetDO drillDone,1;
WaitUntil drillDone = 0;
        MoveL RelTool(Target_500,0,0,-10),v30,z10,DrillTool\WObj:=FakeWing;
        MoveL RelTool(Target_510,0,0,-10),v30,z10,DrillTool\WObj:=FakeWing;
        MoveL Target_510,v30,fine,DrillTool\WObj:=FakeWing;
SetDO drillDone,1;
WaitUntil drillDone = 0;
        MoveL RelTool(Target_510,0,0,-10),v30,z10,DrillTool\WObj:=FakeWing;
        MoveL RelTool(Target_520,0,0,-10),v30,z10,DrillTool\WObj:=FakeWing;
        MoveL Target_520,v30,fine,DrillTool\WObj:=FakeWing;
SetDO drillDone,1;
WaitUntil drillDone = 0;
        MoveL RelTool(Target_520,0,0,-10),v30,z10,DrillTool\WObj:=FakeWing;
        MoveL RelTool(Target_530,0,0,-10),v30,z10,DrillTool\WObj:=FakeWing;
        MoveL Target_530,v30,fine,DrillTool\WObj:=FakeWing;
SetDO drillDone,1;
WaitUntil drillDone = 0;
        MoveL RelTool(Target_530,0,0,-10),v30,z10,DrillTool\WObj:=FakeWing;
        MoveL RelTool(Target_540,0,0,-10),v30,z10,DrillTool\WObj:=FakeWing;
        MoveL Target_540,v30,fine,DrillTool\WObj:=FakeWing;
SetDO drillDone,1;
WaitUntil drillDone = 0;
        MoveL RelTool(Target_540,0,0,-10),v30,z10,DrillTool\WObj:=FakeWing;
        MoveL RelTool(Target_550,0,0,-10),v30,z10,DrillTool\WObj:=FakeWing;
        MoveL Target_550,v30,fine,DrillTool\WObj:=FakeWing;
SetDO drillDone,1;
WaitUntil drillDone = 0;
        MoveL RelTool(Target_550,0,0,-10),v30,z10,DrillTool\WObj:=FakeWing;
        MoveL RelTool(Target_560,0,0,-10),v30,z10,DrillTool\WObj:=FakeWing;
        MoveL Target_560,v30,fine,DrillTool\WObj:=FakeWing;
SetDO drillDone,1;
WaitUntil drillDone = 0;
        MoveL RelTool(Target_560,0,0,-10),v30,z10,DrillTool\WObj:=FakeWing;
        MoveL RelTool(Target_570,0,0,-10),v30,z10,DrillTool\WObj:=FakeWing;
        MoveL Target_570,v30,fine,DrillTool\WObj:=FakeWing;
SetDO drillDone,1;
WaitUntil drillDone = 0;
        MoveL RelTool(Target_570,0,0,-10),v30,z10,DrillTool\WObj:=FakeWing;
        MoveL RelTool(Target_580,0,0,-10),v30,z10,DrillTool\WObj:=FakeWing;
        MoveL Target_580,v30,fine,DrillTool\WObj:=FakeWing;
SetDO drillDone,1;
WaitUntil drillDone = 0;
        MoveL RelTool(Target_580,0,0,-10),v30,z10,DrillTool\WObj:=FakeWing;
        MoveL RelTool(Target_590,0,0,-10),v30,z10,DrillTool\WObj:=FakeWing;
        MoveL Target_590,v30,fine,DrillTool\WObj:=FakeWing;
SetDO drillDone,1;
WaitUntil drillDone = 0;
        MoveL RelTool(Target_590,0,0,-10),v30,z10,DrillTool\WObj:=FakeWing;
        MoveL RelTool(Target_600,0,0,-10),v30,z10,DrillTool\WObj:=FakeWing;
        MoveL Target_600,v30,fine,DrillTool\WObj:=FakeWing;
SetDO drillDone,1;
WaitUntil drillDone = 0;
        MoveL RelTool(Target_600,0,0,-10),v30,z10,DrillTool\WObj:=FakeWing;
        MoveL RelTool(Target_610,0,0,-10),v30,z10,DrillTool\WObj:=FakeWing;
        MoveL Target_610,v30,fine,DrillTool\WObj:=FakeWing;
SetDO drillDone,1;
WaitUntil drillDone = 0;
        MoveL RelTool(Target_610,0,0,-10),v30,z10,DrillTool\WObj:=FakeWing;
        MoveL RelTool(Target_620,0,0,-10),v30,z10,DrillTool\WObj:=FakeWing;
        MoveL Target_620,v30,fine,DrillTool\WObj:=FakeWing;
SetDO drillDone,1;
WaitUntil drillDone = 0;
        MoveL RelTool(Target_620,0,0,-10),v30,z10,DrillTool\WObj:=FakeWing;
        MoveL RelTool(Target_630,0,0,-10),v30,z10,DrillTool\WObj:=FakeWing;
        MoveL Target_630,v30,fine,DrillTool\WObj:=FakeWing;
SetDO drillDone,1;
WaitUntil drillDone = 0;
        MoveL RelTool(Target_630,0,0,-10),v30,z10,DrillTool\WObj:=FakeWing;
        MoveL RelTool(Target_640,0,0,-10),v30,z10,DrillTool\WObj:=FakeWing;
        MoveL Target_640,v30,fine,DrillTool\WObj:=FakeWing;
SetDO drillDone,1;
WaitUntil drillDone = 0;
        MoveL RelTool(Target_640,0,0,-10),v30,z10,DrillTool\WObj:=FakeWing;
        MoveL RelTool(Target_650,0,0,-10),v30,z10,DrillTool\WObj:=FakeWing;
        MoveL Target_650,v30,fine,DrillTool\WObj:=FakeWing;
SetDO drillDone,1;
WaitUntil drillDone = 0;
        MoveL RelTool(Target_650,0,0,-10),v30,z10,DrillTool\WObj:=FakeWing;
        MoveL RelTool(Target_660,0,0,-10),v30,z10,DrillTool\WObj:=FakeWing;
        MoveL Target_660,v30,fine,DrillTool\WObj:=FakeWing;
SetDO drillDone,1;
WaitUntil drillDone = 0;
        MoveL RelTool(Target_660,0,0,-10),v30,z10,DrillTool\WObj:=FakeWing;
        MoveL RelTool(Target_670,0,0,-10),v30,z10,DrillTool\WObj:=FakeWing;
        MoveL Target_670,v30,fine,DrillTool\WObj:=FakeWing;
SetDO drillDone,1;
WaitUntil drillDone = 0;
        MoveL RelTool(Target_670,0,0,-10),v30,z10,DrillTool\WObj:=FakeWing;
        MoveL RelTool(Target_680,0,0,-10),v30,z10,DrillTool\WObj:=FakeWing;
        MoveL Target_680,v30,fine,DrillTool\WObj:=FakeWing;
SetDO drillDone,1;
WaitUntil drillDone = 0;
        MoveL RelTool(Target_680,0,0,-10),v30,z10,DrillTool\WObj:=FakeWing;
        MoveL RelTool(Target_690,0,0,-10),v30,z10,DrillTool\WObj:=FakeWing;
        MoveL Target_690,v30,fine,DrillTool\WObj:=FakeWing;
SetDO drillDone,1;
WaitUntil drillDone = 0;
        MoveL RelTool(Target_690,0,0,-10),v30,z10,DrillTool\WObj:=FakeWing;
        MoveL RelTool(Target_700,0,0,-10),v30,z10,DrillTool\WObj:=FakeWing;
        MoveL Target_700,v30,fine,DrillTool\WObj:=FakeWing;
SetDO drillDone,1;
WaitUntil drillDone = 0;
        MoveL RelTool(Target_700,0,0,-10),v30,z10,DrillTool\WObj:=FakeWing;
        MoveL RelTool(Target_710,0,0,-10),v30,z10,DrillTool\WObj:=FakeWing;
        MoveL Target_710,v30,fine,DrillTool\WObj:=FakeWing;
SetDO drillDone,1;
WaitUntil drillDone = 0;
        MoveL RelTool(Target_710,0,0,-10),v30,z10,DrillTool\WObj:=FakeWing;
        MoveL RelTool(Target_720,0,0,-10),v30,z10,DrillTool\WObj:=FakeWing;
        MoveL Target_720,v30,fine,DrillTool\WObj:=FakeWing;
SetDO drillDone,1;
WaitUntil drillDone = 0;
        MoveL RelTool(Target_720,0,0,-10),v30,z10,DrillTool\WObj:=FakeWing;
        MoveL RelTool(Target_730,0,0,-10),v30,z10,DrillTool\WObj:=FakeWing;
        MoveL Target_730,v30,fine,DrillTool\WObj:=FakeWing;
SetDO drillDone,1;
WaitUntil drillDone = 0;
        MoveL RelTool(Target_730,0,0,-10),v30,z10,DrillTool\WObj:=FakeWing;
        MoveL RelTool(Target_740,0,0,-10),v30,z10,DrillTool\WObj:=FakeWing;
        MoveL Target_740,v30,fine,DrillTool\WObj:=FakeWing;
SetDO drillDone,1;
WaitUntil drillDone = 0;
        MoveL RelTool(Target_740,0,0,-10),v30,z10,DrillTool\WObj:=FakeWing;
        MoveL RelTool(Target_750,0,0,-10),v30,z10,DrillTool\WObj:=FakeWing;
        MoveL Target_750,v30,fine,DrillTool\WObj:=FakeWing;
SetDO drillDone,1;
WaitUntil drillDone = 0;
        MoveL RelTool(Target_750,0,0,-10),v30,z10,DrillTool\WObj:=FakeWing;
        MoveL RelTool(Target_760,0,0,-10),v30,z10,DrillTool\WObj:=FakeWing;
        MoveL Target_760,v30,fine,DrillTool\WObj:=FakeWing;
SetDO drillDone,1;
WaitUntil drillDone = 0;
        MoveL RelTool(Target_760,0,0,-10),v30,z10,DrillTool\WObj:=FakeWing;
        MoveL RelTool(Target_770,0,0,-10),v30,z10,DrillTool\WObj:=FakeWing;
        MoveL Target_770,v30,fine,DrillTool\WObj:=FakeWing;
SetDO drillDone,1;
WaitUntil drillDone = 0;
        MoveL RelTool(Target_770,0,0,-10),v30,z10,DrillTool\WObj:=FakeWing;
        MoveL RelTool(Target_780,0,0,-10),v30,z10,DrillTool\WObj:=FakeWing;
        MoveL Target_780,v30,fine,DrillTool\WObj:=FakeWing;
SetDO drillDone,1;
WaitUntil drillDone = 0;
        MoveL RelTool(Target_780,0,0,-10),v30,z10,DrillTool\WObj:=FakeWing;
        MoveL RelTool(Target_790,0,0,-10),v30,z10,DrillTool\WObj:=FakeWing;
        MoveL Target_790,v30,fine,DrillTool\WObj:=FakeWing;
SetDO drillDone,1;
WaitUntil drillDone = 0;
        MoveL RelTool(Target_790,0,0,-10),v30,z10,DrillTool\WObj:=FakeWing;
        MoveL RelTool(Target_800,0,0,-10),v30,z10,DrillTool\WObj:=FakeWing;
        MoveL Target_800,v30,fine,DrillTool\WObj:=FakeWing;
SetDO drillDone,1;
WaitUntil drillDone = 0;
        MoveL RelTool(Target_800,0,0,-10),v30,z10,DrillTool\WObj:=FakeWing;
        MoveL RelTool(Target_810,0,0,-10),v30,z10,DrillTool\WObj:=FakeWing;
        MoveL Target_810,v30,fine,DrillTool\WObj:=FakeWing;
SetDO drillDone,1;
WaitUntil drillDone = 0;
        MoveL RelTool(Target_810,0,0,-10),v30,z10,DrillTool\WObj:=FakeWing;
        MoveL RelTool(Target_820,0,0,-10),v30,z10,DrillTool\WObj:=FakeWing;
        MoveL Target_820,v30,fine,DrillTool\WObj:=FakeWing;
SetDO drillDone,1;
WaitUntil drillDone = 0;
        MoveL RelTool(Target_820,0,0,-10),v30,z10,DrillTool\WObj:=FakeWing;
        MoveL RelTool(Target_830,0,0,-10),v30,z10,DrillTool\WObj:=FakeWing;
        MoveL Target_830,v30,fine,DrillTool\WObj:=FakeWing;
SetDO drillDone,1;
WaitUntil drillDone = 0;
        MoveL RelTool(Target_830,0,0,-10),v30,z10,DrillTool\WObj:=FakeWing;
        MoveL RelTool(Target_840,0,0,-10),v30,z10,DrillTool\WObj:=FakeWing;
        MoveL Target_840,v30,fine,DrillTool\WObj:=FakeWing;
SetDO drillDone,1;
WaitUntil drillDone = 0;
        MoveL RelTool(Target_840,0,0,-10),v30,z10,DrillTool\WObj:=FakeWing;
        MoveL RelTool(Target_850,0,0,-10),v30,z10,DrillTool\WObj:=FakeWing;
        MoveL Target_850,v30,fine,DrillTool\WObj:=FakeWing;
SetDO drillDone,1;
WaitUntil drillDone = 0;
        MoveL RelTool(Target_850,0,0,-10),v30,z10,DrillTool\WObj:=FakeWing;
        MoveL RelTool(Target_860,0,0,-10),v30,z10,DrillTool\WObj:=FakeWing;
        MoveL Target_860,v30,fine,DrillTool\WObj:=FakeWing;
SetDO drillDone,1;
WaitUntil drillDone = 0;
        MoveL RelTool(Target_860,0,0,-10),v30,z10,DrillTool\WObj:=FakeWing;
        MoveL RelTool(Target_870,0,0,-10),v30,z10,DrillTool\WObj:=FakeWing;
        MoveL Target_870,v30,fine,DrillTool\WObj:=FakeWing;
SetDO drillDone,1;
WaitUntil drillDone = 0;
        MoveL RelTool(Target_870,0,0,-10),v30,z10,DrillTool\WObj:=FakeWing;
        MoveL RelTool(Target_880,0,0,-10),v30,z10,DrillTool\WObj:=FakeWing;
        MoveL Target_880,v30,fine,DrillTool\WObj:=FakeWing;
SetDO drillDone,1;
WaitUntil drillDone = 0;
        MoveL RelTool(Target_880,0,0,-10),v30,z10,DrillTool\WObj:=FakeWing;
        MoveL RelTool(Target_890,0,0,-10),v30,z10,DrillTool\WObj:=FakeWing;
        MoveL Target_890,v30,fine,DrillTool\WObj:=FakeWing;
SetDO drillDone,1;
WaitUntil drillDone = 0;
        MoveL RelTool(Target_890,0,0,-10),v30,z10,DrillTool\WObj:=FakeWing;
        MoveL RelTool(Target_900,0,0,-10),v30,z10,DrillTool\WObj:=FakeWing;
        MoveL Target_900,v30,fine,DrillTool\WObj:=FakeWing;
SetDO drillDone,1;
WaitUntil drillDone = 0;
        MoveL RelTool(Target_900,0,0,-10),v30,z10,DrillTool\WObj:=FakeWing;
        MoveL RelTool(Target_910,0,0,-10),v30,z10,DrillTool\WObj:=FakeWing;
        MoveL Target_910,v30,fine,DrillTool\WObj:=FakeWing;
SetDO drillDone,1;
WaitUntil drillDone = 0;
        MoveL RelTool(Target_910,0,0,-10),v30,z10,DrillTool\WObj:=FakeWing;
        MoveL RelTool(Target_920,0,0,-10),v30,z10,DrillTool\WObj:=FakeWing;
        MoveL Target_920,v30,fine,DrillTool\WObj:=FakeWing;
SetDO drillDone,1;
WaitUntil drillDone = 0;
        MoveL RelTool(Target_920,0,0,-10),v30,z10,DrillTool\WObj:=FakeWing;
        MoveL RelTool(Target_930,0,0,-10),v30,z10,DrillTool\WObj:=FakeWing;
        MoveL Target_930,v30,fine,DrillTool\WObj:=FakeWing;
SetDO drillDone,1;
WaitUntil drillDone = 0;
        MoveL RelTool(Target_930,0,0,-10),v30,z10,DrillTool\WObj:=FakeWing;
        MoveL RelTool(Target_940,0,0,-10),v30,z10,DrillTool\WObj:=FakeWing;
        MoveL Target_940,v30,fine,DrillTool\WObj:=FakeWing;
SetDO drillDone,1;
WaitUntil drillDone = 0;
        MoveL RelTool(Target_940,0,0,-10),v30,z10,DrillTool\WObj:=FakeWing;
        MoveL RelTool(Target_950,0,0,-10),v30,z10,DrillTool\WObj:=FakeWing;
        MoveL Target_950,v30,fine,DrillTool\WObj:=FakeWing;
SetDO drillDone,1;
WaitUntil drillDone = 0;
        MoveL RelTool(Target_950,0,0,-10),v30,z10,DrillTool\WObj:=FakeWing;
        MoveL RelTool(Target_960,0,0,-10),v30,z10,DrillTool\WObj:=FakeWing;
        MoveL Target_960,v30,fine,DrillTool\WObj:=FakeWing;
SetDO drillDone,1;
WaitUntil drillDone = 0;
        MoveL RelTool(Target_960,0,0,-10),v30,z10,DrillTool\WObj:=FakeWing;
        MoveL RelTool(Target_970,0,0,-10),v30,z10,DrillTool\WObj:=FakeWing;
        MoveL Target_970,v30,fine,DrillTool\WObj:=FakeWing;
SetDO drillDone,1;
WaitUntil drillDone = 0;
        MoveL RelTool(Target_970,0,0,-10),v30,z10,DrillTool\WObj:=FakeWing;
        MoveL RelTool(Target_980,0,0,-10),v30,z10,DrillTool\WObj:=FakeWing;
        MoveL Target_980,v30,fine,DrillTool\WObj:=FakeWing;
SetDO drillDone,1;
WaitUntil drillDone = 0;
        MoveL RelTool(Target_980,0,0,-10),v30,z10,DrillTool\WObj:=FakeWing;
        MoveL RelTool(Target_990,0,0,-10),v30,z10,DrillTool\WObj:=FakeWing;
        MoveL Target_990,v30,fine,DrillTool\WObj:=FakeWing;
SetDO drillDone,1;
WaitUntil drillDone = 0;
        MoveL RelTool(Target_990,0,0,-10),v30,z10,DrillTool\WObj:=FakeWing;
        MoveL RelTool(Target_1000,0,0,-10),v30,z10,DrillTool\WObj:=FakeWing;
        MoveL Target_1000,v30,fine,DrillTool\WObj:=FakeWing;
SetDO drillDone,1;
WaitUntil drillDone = 0;
        MoveL RelTool(Target_1000,0,0,-10),v30,z10,DrillTool\WObj:=FakeWing;
        MoveL RelTool(Target_1010,0,0,-10),v30,z10,DrillTool\WObj:=FakeWing;
        MoveL Target_1010,v30,fine,DrillTool\WObj:=FakeWing;
SetDO drillDone,1;
WaitUntil drillDone = 0;
        MoveL RelTool(Target_1010,0,0,-10),v30,z10,DrillTool\WObj:=FakeWing;
        MoveL RelTool(Target_1020,0,0,-10),v30,z10,DrillTool\WObj:=FakeWing;
        MoveL Target_1020,v30,fine,DrillTool\WObj:=FakeWing;
SetDO drillDone,1;
WaitUntil drillDone = 0;
        MoveL RelTool(Target_1020,0,0,-10),v30,z10,DrillTool\WObj:=FakeWing;
        MoveL RelTool(Target_1030,0,0,-10),v30,z10,DrillTool\WObj:=FakeWing;
        MoveL Target_1030,v30,fine,DrillTool\WObj:=FakeWing;
SetDO drillDone,1;
WaitUntil drillDone = 0;
        MoveL RelTool(Target_1030,0,0,-10),v30,z10,DrillTool\WObj:=FakeWing;
        MoveL RelTool(Target_1040,0,0,-10),v30,z10,DrillTool\WObj:=FakeWing;
        MoveL Target_1040,v30,fine,DrillTool\WObj:=FakeWing;
SetDO drillDone,1;
WaitUntil drillDone = 0;
        MoveL RelTool(Target_1040,0,0,-10),v30,z10,DrillTool\WObj:=FakeWing;
        MoveL RelTool(Target_1050,0,0,-10),v30,z10,DrillTool\WObj:=FakeWing;
        MoveL Target_1050,v30,fine,DrillTool\WObj:=FakeWing;
SetDO drillDone,1;
WaitUntil drillDone = 0;
        MoveL RelTool(Target_1050,0,0,-10),v30,z10,DrillTool\WObj:=FakeWing;
        MoveL RelTool(Target_1060,0,0,-10),v30,z10,DrillTool\WObj:=FakeWing;
        MoveL Target_1060,v30,fine,DrillTool\WObj:=FakeWing;
SetDO drillDone,1;
WaitUntil drillDone = 0;
        MoveL RelTool(Target_1060,0,0,-10),v30,z10,DrillTool\WObj:=FakeWing;
        MoveL RelTool(Target_1070,0,0,-10),v30,z10,DrillTool\WObj:=FakeWing;
        MoveL Target_1070,v30,fine,DrillTool\WObj:=FakeWing;
SetDO drillDone,1;
WaitUntil drillDone = 0;
        MoveL RelTool(Target_1070,0,0,-10),v30,z10,DrillTool\WObj:=FakeWing;
        MoveL RelTool(Target_1080,0,0,-10),v30,z10,DrillTool\WObj:=FakeWing;
        MoveL Target_1080,v30,fine,DrillTool\WObj:=FakeWing;
SetDO drillDone,1;
WaitUntil drillDone = 0;
        MoveL RelTool(Target_1080,0,0,-10),v30,z10,DrillTool\WObj:=FakeWing;
        MoveL RelTool(Target_1090,0,0,-10),v30,z10,DrillTool\WObj:=FakeWing;
        MoveL Target_1090,v30,fine,DrillTool\WObj:=FakeWing;
SetDO drillDone,1;
WaitUntil drillDone = 0;
        MoveL RelTool(Target_1090,0,0,-10),v30,z10,DrillTool\WObj:=FakeWing;
        MoveL RelTool(Target_1100,0,0,-10),v30,z10,DrillTool\WObj:=FakeWing;
        MoveL Target_1100,v30,fine,DrillTool\WObj:=FakeWing;
SetDO drillDone,1;
WaitUntil drillDone = 0;
        MoveL RelTool(Target_1100,0,0,-10),v30,z10,DrillTool\WObj:=FakeWing;
        MoveL RelTool(Target_1110,0,0,-10),v30,z10,DrillTool\WObj:=FakeWing;
        MoveL Target_1110,v30,fine,DrillTool\WObj:=FakeWing;
SetDO drillDone,1;
WaitUntil drillDone = 0;
        MoveL RelTool(Target_1110,0,0,-10),v30,z10,DrillTool\WObj:=FakeWing;
        MoveL RelTool(Target_1120,0,0,-10),v30,z10,DrillTool\WObj:=FakeWing;
        MoveL Target_1120,v30,fine,DrillTool\WObj:=FakeWing;
SetDO drillDone,1;
WaitUntil drillDone = 0;
        MoveL RelTool(Target_1120,0,0,-10),v30,z10,DrillTool\WObj:=FakeWing;
        MoveL RelTool(Target_1130,0,0,-10),v30,z10,DrillTool\WObj:=FakeWing;
        MoveL Target_1130,v30,fine,DrillTool\WObj:=FakeWing;
SetDO drillDone,1;
WaitUntil drillDone = 0;
        MoveL RelTool(Target_1130,0,0,-10),v30,z10,DrillTool\WObj:=FakeWing;
        MoveL RelTool(Target_1140,0,0,-10),v30,z10,DrillTool\WObj:=FakeWing;
        MoveL Target_1140,v30,fine,DrillTool\WObj:=FakeWing;
SetDO drillDone,1;
WaitUntil drillDone = 0;
        MoveL RelTool(Target_1140,0,0,-10),v30,z10,DrillTool\WObj:=FakeWing;
        MoveL RelTool(Target_1150,0,0,-10),v30,z10,DrillTool\WObj:=FakeWing;
        MoveL Target_1150,v30,fine,DrillTool\WObj:=FakeWing;
SetDO drillDone,1;
WaitUntil drillDone = 0;
        MoveL RelTool(Target_1150,0,0,-10),v30,z10,DrillTool\WObj:=FakeWing;
        MoveL RelTool(Target_1160,0,0,-10),v30,z10,DrillTool\WObj:=FakeWing;
        MoveL Target_1160,v30,fine,DrillTool\WObj:=FakeWing;
SetDO drillDone,1;
WaitUntil drillDone = 0;
        MoveL RelTool(Target_1160,0,0,-10),v30,z10,DrillTool\WObj:=FakeWing;
        MoveL RelTool(Target_1170,0,0,-10),v30,z10,DrillTool\WObj:=FakeWing;
        MoveL Target_1170,v30,fine,DrillTool\WObj:=FakeWing;
SetDO drillDone,1;
WaitUntil drillDone = 0;
        MoveL RelTool(Target_1170,0,0,-10),v30,z10,DrillTool\WObj:=FakeWing;
        MoveL RelTool(Target_1180,0,0,-10),v30,z10,DrillTool\WObj:=FakeWing;
        MoveL Target_1180,v30,fine,DrillTool\WObj:=FakeWing;
SetDO drillDone,1;
WaitUntil drillDone = 0;
        MoveL RelTool(Target_1180,0,0,-10),v30,z10,DrillTool\WObj:=FakeWing;
        MoveL RelTool(Target_1190,0,0,-10),v30,z10,DrillTool\WObj:=FakeWing;
        MoveL Target_1190,v30,fine,DrillTool\WObj:=FakeWing;
SetDO drillDone,1;
WaitUntil drillDone = 0;
        MoveL RelTool(Target_1190,0,0,-10),v30,z10,DrillTool\WObj:=FakeWing;
        MoveL RelTool(Target_1200,0,0,-10),v30,z10,DrillTool\WObj:=FakeWing;
        MoveL Target_1200,v30,fine,DrillTool\WObj:=FakeWing;
SetDO drillDone,1;
WaitUntil drillDone = 0;
        MoveL RelTool(Target_1200,0,0,-10),v30,z10,DrillTool\WObj:=FakeWing;
        MoveL RelTool(Target_1210,0,0,-10),v30,z10,DrillTool\WObj:=FakeWing;
        MoveL Target_1210,v30,fine,DrillTool\WObj:=FakeWing;
SetDO drillDone,1;
WaitUntil drillDone = 0;
        MoveL RelTool(Target_1210,0,0,-10),v30,z10,DrillTool\WObj:=FakeWing;
        MoveL RelTool(Target_1220,0,0,-10),v30,z10,DrillTool\WObj:=FakeWing;
        MoveL Target_1220,v30,fine,DrillTool\WObj:=FakeWing;
SetDO drillDone,1;
WaitUntil drillDone = 0;
        MoveL RelTool(Target_1220,0,0,-10),v30,z10,DrillTool\WObj:=FakeWing;
        MoveL RelTool(Target_1230,0,0,-10),v30,z10,DrillTool\WObj:=FakeWing;
        MoveL Target_1230,v30,fine,DrillTool\WObj:=FakeWing;
SetDO drillDone,1;
WaitUntil drillDone = 0;
        MoveL RelTool(Target_1230,0,0,-10),v30,z10,DrillTool\WObj:=FakeWing;
        MoveL RelTool(Target_1240,0,0,-10),v30,z10,DrillTool\WObj:=FakeWing;
        MoveL Target_1240,v30,fine,DrillTool\WObj:=FakeWing;
SetDO drillDone,1;
WaitUntil drillDone = 0;
        MoveL RelTool(Target_1240,0,0,-10),v30,z10,DrillTool\WObj:=FakeWing;
        MoveL RelTool(Target_1250,0,0,-10),v30,z10,DrillTool\WObj:=FakeWing;
        MoveL Target_1250,v30,fine,DrillTool\WObj:=FakeWing;
SetDO drillDone,1;
WaitUntil drillDone = 0;
        MoveL RelTool(Target_1250,0,0,-10),v30,z10,DrillTool\WObj:=FakeWing;
        MoveL RelTool(Target_1260,0,0,-10),v30,z10,DrillTool\WObj:=FakeWing;
        MoveL Target_1260,v30,fine,DrillTool\WObj:=FakeWing;
SetDO drillDone,1;
WaitUntil drillDone = 0;
        MoveL RelTool(Target_1260,0,0,-10),v30,z10,DrillTool\WObj:=FakeWing;
        MoveL RelTool(Target_1270,0,0,-10),v30,z10,DrillTool\WObj:=FakeWing;
        MoveL Target_1270,v30,fine,DrillTool\WObj:=FakeWing;
SetDO drillDone,1;
WaitUntil drillDone = 0;
        MoveL RelTool(Target_1270,0,0,-10),v30,z10,DrillTool\WObj:=FakeWing;
        MoveL RelTool(Target_1280,0,0,-10),v30,z10,DrillTool\WObj:=FakeWing;
        MoveL Target_1280,v30,fine,DrillTool\WObj:=FakeWing;
SetDO drillDone,1;
WaitUntil drillDone = 0;
        MoveL RelTool(Target_1280,0,0,-10),v30,z10,DrillTool\WObj:=FakeWing;
        MoveL RelTool(Target_1290,0,0,-10),v30,z10,DrillTool\WObj:=FakeWing;
        MoveL Target_1290,v30,fine,DrillTool\WObj:=FakeWing;
SetDO drillDone,1;
WaitUntil drillDone = 0;
        MoveL RelTool(Target_1290,0,0,-10),v30,z10,DrillTool\WObj:=FakeWing;
        MoveL RelTool(Target_1300,0,0,-10),v30,z10,DrillTool\WObj:=FakeWing;
        MoveL Target_1300,v30,fine,DrillTool\WObj:=FakeWing;
SetDO drillDone,1;
WaitUntil drillDone = 0;
        MoveL RelTool(Target_1300,0,0,-10),v30,z10,DrillTool\WObj:=FakeWing;
        MoveL RelTool(Target_1310,0,0,-10),v30,z10,DrillTool\WObj:=FakeWing;
        MoveL Target_1310,v30,fine,DrillTool\WObj:=FakeWing;
SetDO drillDone,1;
WaitUntil drillDone = 0;
        MoveL RelTool(Target_1310,0,0,-10),v30,z10,DrillTool\WObj:=FakeWing;
        MoveL RelTool(Target_1320,0,0,-10),v30,z10,DrillTool\WObj:=FakeWing;
        MoveL Target_1320,v30,fine,DrillTool\WObj:=FakeWing;
SetDO drillDone,1;
WaitUntil drillDone = 0;
        MoveL RelTool(Target_1320,0,0,-10),v30,z10,DrillTool\WObj:=FakeWing;
        MoveL RelTool(Target_1330,0,0,-10),v30,z10,DrillTool\WObj:=FakeWing;
        MoveL Target_1330,v30,fine,DrillTool\WObj:=FakeWing;
SetDO drillDone,1;
WaitUntil drillDone = 0;
        MoveL RelTool(Target_1330,0,0,-10),v30,z10,DrillTool\WObj:=FakeWing;
        MoveL RelTool(Target_1340,0,0,-10),v30,z10,DrillTool\WObj:=FakeWing;
        MoveL Target_1340,v30,fine,DrillTool\WObj:=FakeWing;
SetDO drillDone,1;
WaitUntil drillDone = 0;
        MoveL RelTool(Target_1340,0,0,-10),v30,z10,DrillTool\WObj:=FakeWing;
        MoveL RelTool(Target_1350,0,0,-10),v30,z10,DrillTool\WObj:=FakeWing;
        MoveL Target_1350,v30,fine,DrillTool\WObj:=FakeWing;
SetDO drillDone,1;
WaitUntil drillDone = 0;
        MoveL RelTool(Target_1350,0,0,-10),v30,z10,DrillTool\WObj:=FakeWing;
        MoveL RelTool(Target_1360,0,0,-10),v30,z10,DrillTool\WObj:=FakeWing;
        MoveL Target_1360,v30,fine,DrillTool\WObj:=FakeWing;
SetDO drillDone,1;
WaitUntil drillDone = 0;
        MoveL RelTool(Target_1360,0,0,-10),v30,z10,DrillTool\WObj:=FakeWing;
        MoveL RelTool(Target_1370,0,0,-10),v30,z10,DrillTool\WObj:=FakeWing;
        MoveL Target_1370,v30,fine,DrillTool\WObj:=FakeWing;
SetDO drillDone,1;
WaitUntil drillDone = 0;
        MoveL RelTool(Target_1370,0,0,-10),v30,z10,DrillTool\WObj:=FakeWing;
        MoveL RelTool(Target_1380,0,0,-10),v30,z10,DrillTool\WObj:=FakeWing;
        MoveL Target_1380,v30,fine,DrillTool\WObj:=FakeWing;
SetDO drillDone,1;
WaitUntil drillDone = 0;
        MoveL RelTool(Target_1380,0,0,-10),v30,z10,DrillTool\WObj:=FakeWing;
        MoveL RelTool(Target_1390,0,0,-10),v30,z10,DrillTool\WObj:=FakeWing;
        MoveL Target_1390,v30,fine,DrillTool\WObj:=FakeWing;
SetDO drillDone,1;
WaitUntil drillDone = 0;
        MoveL RelTool(Target_1390,0,0,-10),v30,z10,DrillTool\WObj:=FakeWing;
        MoveL RelTool(Target_1400,0,0,-10),v30,z10,DrillTool\WObj:=FakeWing;
        MoveL Target_1400,v30,fine,DrillTool\WObj:=FakeWing;
SetDO drillDone,1;
WaitUntil drillDone = 0;
        MoveL RelTool(Target_1400,0,0,-10),v30,z10,DrillTool\WObj:=FakeWing;
        MoveL RelTool(Target_1410,0,0,-10),v30,z10,DrillTool\WObj:=FakeWing;
        MoveL Target_1410,v30,fine,DrillTool\WObj:=FakeWing;
SetDO drillDone,1;
WaitUntil drillDone = 0;
        MoveL RelTool(Target_1410,0,0,-10),v30,z10,DrillTool\WObj:=FakeWing;
        MoveL RelTool(Target_1420,0,0,-10),v30,z10,DrillTool\WObj:=FakeWing;
        MoveL Target_1420,v30,fine,DrillTool\WObj:=FakeWing;
SetDO drillDone,1;
WaitUntil drillDone = 0;
        MoveL RelTool(Target_1420,0,0,-10),v30,z10,DrillTool\WObj:=FakeWing;
        MoveL RelTool(Target_1430,0,0,-10),v30,z10,DrillTool\WObj:=FakeWing;
        MoveL Target_1430,v30,fine,DrillTool\WObj:=FakeWing;
SetDO drillDone,1;
WaitUntil drillDone = 0;
        MoveL RelTool(Target_1430,0,0,-10),v30,z10,DrillTool\WObj:=FakeWing;
        MoveL RelTool(Target_1440,0,0,-10),v30,z10,DrillTool\WObj:=FakeWing;
        MoveL Target_1440,v30,fine,DrillTool\WObj:=FakeWing;
SetDO drillDone,1;
WaitUntil drillDone = 0;
        MoveL RelTool(Target_1440,0,0,-10),v30,z10,DrillTool\WObj:=FakeWing;
        MoveL RelTool(Target_1450,0,0,-10),v30,z10,DrillTool\WObj:=FakeWing;
        MoveL Target_1450,v30,fine,DrillTool\WObj:=FakeWing;
SetDO drillDone,1;
WaitUntil drillDone = 0;
        MoveL RelTool(Target_1450,0,0,-10),v30,z10,DrillTool\WObj:=FakeWing;
        MoveL RelTool(Target_1460,0,0,-10),v30,z10,DrillTool\WObj:=FakeWing;
        MoveL Target_1460,v30,fine,DrillTool\WObj:=FakeWing;
SetDO drillDone,1;
WaitUntil drillDone = 0;
        MoveL RelTool(Target_1460,0,0,-10),v30,z10,DrillTool\WObj:=FakeWing;
        MoveL RelTool(Target_1470,0,0,-10),v30,z10,DrillTool\WObj:=FakeWing;
        MoveL Target_1470,v30,fine,DrillTool\WObj:=FakeWing;
SetDO drillDone,1;
WaitUntil drillDone = 0;
        MoveL RelTool(Target_1470,0,0,-10),v30,z10,DrillTool\WObj:=FakeWing;
        MoveL RelTool(Target_1480,0,0,-10),v30,z10,DrillTool\WObj:=FakeWing;
        MoveL Target_1480,v30,fine,DrillTool\WObj:=FakeWing;
SetDO drillDone,1;
WaitUntil drillDone = 0;
        MoveL RelTool(Target_1480,0,0,-10),v30,z10,DrillTool\WObj:=FakeWing;
        MoveL RelTool(Target_1490,0,0,-10),v30,z10,DrillTool\WObj:=FakeWing;
        MoveL Target_1490,v30,fine,DrillTool\WObj:=FakeWing;
SetDO drillDone,1;
WaitUntil drillDone = 0;
        MoveL RelTool(Target_1490,0,0,-10),v30,z10,DrillTool\WObj:=FakeWing;
        MoveL RelTool(Target_1500,0,0,-10),v30,z10,DrillTool\WObj:=FakeWing;
        MoveL Target_1500,v30,fine,DrillTool\WObj:=FakeWing;
SetDO drillDone,1;
WaitUntil drillDone = 0;
        MoveL RelTool(Target_1500,0,0,-10),v30,z10,DrillTool\WObj:=FakeWing;
        MoveL RelTool(Target_1510,0,0,-10),v30,z10,DrillTool\WObj:=FakeWing;
        MoveL Target_1510,v30,fine,DrillTool\WObj:=FakeWing;
SetDO drillDone,1;
WaitUntil drillDone = 0;
        MoveL RelTool(Target_1510,0,0,-10),v30,z10,DrillTool\WObj:=FakeWing;
        MoveL RelTool(Target_1520,0,0,-10),v30,z10,DrillTool\WObj:=FakeWing;
        MoveL Target_1520,v30,fine,DrillTool\WObj:=FakeWing;
SetDO drillDone,1;
WaitUntil drillDone = 0;
        MoveL RelTool(Target_1520,0,0,-10),v30,z10,DrillTool\WObj:=FakeWing;
        MoveL RelTool(Target_1530,0,0,-10),v30,z10,DrillTool\WObj:=FakeWing;
        MoveL Target_1530,v30,fine,DrillTool\WObj:=FakeWing;
SetDO drillDone,1;
WaitUntil drillDone = 0;
        MoveL RelTool(Target_1530,0,0,-10),v30,z10,DrillTool\WObj:=FakeWing;
        MoveL RelTool(Target_1540,0,0,-10),v30,z10,DrillTool\WObj:=FakeWing;
        MoveL Target_1540,v30,fine,DrillTool\WObj:=FakeWing;
SetDO drillDone,1;
WaitUntil drillDone = 0;
        MoveL RelTool(Target_1540,0,0,-10),v30,z10,DrillTool\WObj:=FakeWing;
        MoveL RelTool(Target_1550,0,0,-10),v30,z10,DrillTool\WObj:=FakeWing;
        MoveL Target_1550,v30,fine,DrillTool\WObj:=FakeWing;
SetDO drillDone,1;
WaitUntil drillDone = 0;
        MoveL RelTool(Target_1550,0,0,-10),v30,z10,DrillTool\WObj:=FakeWing;
        MoveL RelTool(Target_1560,0,0,-10),v30,z10,DrillTool\WObj:=FakeWing;
        MoveL Target_1560,v30,fine,DrillTool\WObj:=FakeWing;
SetDO drillDone,1;
WaitUntil drillDone = 0;
        MoveL RelTool(Target_1560,0,0,-10),v30,z10,DrillTool\WObj:=FakeWing;
        MoveL RelTool(Target_1570,0,0,-10),v30,z10,DrillTool\WObj:=FakeWing;
        MoveL Target_1570,v30,fine,DrillTool\WObj:=FakeWing;
SetDO drillDone,1;
WaitUntil drillDone = 0;
        MoveL RelTool(Target_1570,0,0,-10),v30,z10,DrillTool\WObj:=FakeWing;
        MoveL RelTool(Target_1580,0,0,-10),v30,z10,DrillTool\WObj:=FakeWing;
        MoveL Target_1580,v30,fine,DrillTool\WObj:=FakeWing;
SetDO drillDone,1;
WaitUntil drillDone = 0;
        MoveL RelTool(Target_1580,0,0,-10),v30,z10,DrillTool\WObj:=FakeWing;
        MoveL RelTool(Target_1590,0,0,-10),v30,z10,DrillTool\WObj:=FakeWing;
        MoveL Target_1590,v30,fine,DrillTool\WObj:=FakeWing;
SetDO drillDone,1;
WaitUntil drillDone = 0;
        MoveL RelTool(Target_1590,0,0,-10),v30,z10,DrillTool\WObj:=FakeWing;
        MoveL RelTool(Target_1600,0,0,-10),v30,z10,DrillTool\WObj:=FakeWing;
        MoveL Target_1600,v30,fine,DrillTool\WObj:=FakeWing;
SetDO drillDone,1;
WaitUntil drillDone = 0;
        MoveL RelTool(Target_1600,0,0,-10),v30,z10,DrillTool\WObj:=FakeWing;
        MoveL RelTool(Target_1610,0,0,-10),v30,z10,DrillTool\WObj:=FakeWing;
        MoveL Target_1610,v30,fine,DrillTool\WObj:=FakeWing;
SetDO drillDone,1;
WaitUntil drillDone = 0;
        MoveL RelTool(Target_1610,0,0,-10),v30,z10,DrillTool\WObj:=FakeWing;
        MoveL RelTool(Target_1620,0,0,-10),v30,z10,DrillTool\WObj:=FakeWing;
        MoveL Target_1620,v30,fine,DrillTool\WObj:=FakeWing;
SetDO drillDone,1;
WaitUntil drillDone = 0;
        MoveL RelTool(Target_1620,0,0,-10),v30,z10,DrillTool\WObj:=FakeWing;
        MoveL RelTool(Target_1630,0,0,-10),v30,z10,DrillTool\WObj:=FakeWing;
        MoveL Target_1630,v30,fine,DrillTool\WObj:=FakeWing;
SetDO drillDone,1;
WaitUntil drillDone = 0;
        MoveL RelTool(Target_1630,0,0,-10),v30,z10,DrillTool\WObj:=FakeWing;
        MoveL RelTool(Target_1640,0,0,-10),v30,z10,DrillTool\WObj:=FakeWing;
        MoveL Target_1640,v30,fine,DrillTool\WObj:=FakeWing;
SetDO drillDone,1;
WaitUntil drillDone = 0;
        MoveL RelTool(Target_1640,0,0,-10),v30,z10,DrillTool\WObj:=FakeWing;
        MoveL RelTool(Target_1650,0,0,-10),v30,z10,DrillTool\WObj:=FakeWing;
        MoveL Target_1650,v30,fine,DrillTool\WObj:=FakeWing;
SetDO drillDone,1;
WaitUntil drillDone = 0;
        MoveL RelTool(Target_1650,0,0,-10),v30,z10,DrillTool\WObj:=FakeWing;
        MoveL RelTool(Target_1660,0,0,-10),v30,z10,DrillTool\WObj:=FakeWing;
        MoveL Target_1660,v30,fine,DrillTool\WObj:=FakeWing;
SetDO drillDone,1;
WaitUntil drillDone = 0;
        MoveL RelTool(Target_1660,0,0,-10),v30,z10,DrillTool\WObj:=FakeWing;
        MoveL RelTool(Target_1670,0,0,-10),v30,z10,DrillTool\WObj:=FakeWing;
        MoveL Target_1670,v30,fine,DrillTool\WObj:=FakeWing;
SetDO drillDone,1;
WaitUntil drillDone = 0;
        MoveL RelTool(Target_1670,0,0,-10),v30,z10,DrillTool\WObj:=FakeWing;
        MoveL RelTool(Target_1680,0,0,-10),v30,z10,DrillTool\WObj:=FakeWing;
        MoveL Target_1680,v30,fine,DrillTool\WObj:=FakeWing;
SetDO drillDone,1;
WaitUntil drillDone = 0;
        MoveL RelTool(Target_1680,0,0,-10),v30,z10,DrillTool\WObj:=FakeWing;
        MoveL RelTool(Target_1690,0,0,-10),v30,z10,DrillTool\WObj:=FakeWing;
        MoveL Target_1690,v30,fine,DrillTool\WObj:=FakeWing;
SetDO drillDone,1;
WaitUntil drillDone = 0;
        MoveL RelTool(Target_1690,0,0,-10),v30,z10,DrillTool\WObj:=FakeWing;
        MoveL RelTool(Target_1700,0,0,-10),v30,z10,DrillTool\WObj:=FakeWing;
        MoveL Target_1700,v30,fine,DrillTool\WObj:=FakeWing;
SetDO drillDone,1;
WaitUntil drillDone = 0;
        MoveL RelTool(Target_1700,0,0,-10),v30,z10,DrillTool\WObj:=FakeWing;
        MoveL RelTool(Target_1710,0,0,-10),v30,z10,DrillTool\WObj:=FakeWing;
        MoveL Target_1710,v30,fine,DrillTool\WObj:=FakeWing;
SetDO drillDone,1;
WaitUntil drillDone = 0;
        MoveL RelTool(Target_1710,0,0,-10),v30,z10,DrillTool\WObj:=FakeWing;
        MoveL RelTool(Target_1720,0,0,-10),v30,z10,DrillTool\WObj:=FakeWing;
        MoveL Target_1720,v30,fine,DrillTool\WObj:=FakeWing;
SetDO drillDone,1;
WaitUntil drillDone = 0;
        MoveL RelTool(Target_1720,0,0,-10),v30,z10,DrillTool\WObj:=FakeWing;
        MoveL RelTool(Target_1730,0,0,-10),v30,z10,DrillTool\WObj:=FakeWing;
        MoveL Target_1730,v30,fine,DrillTool\WObj:=FakeWing;
SetDO drillDone,1;
WaitUntil drillDone = 0;
        MoveL RelTool(Target_1730,0,0,-10),v30,z10,DrillTool\WObj:=FakeWing;
        MoveL RelTool(Target_1740,0,0,-10),v30,z10,DrillTool\WObj:=FakeWing;
        MoveL Target_1740,v30,fine,DrillTool\WObj:=FakeWing;
SetDO drillDone,1;
WaitUntil drillDone = 0;
        MoveL RelTool(Target_1740,0,0,-10),v30,z10,DrillTool\WObj:=FakeWing;
        MoveL RelTool(Target_1750,0,0,-10),v30,z10,DrillTool\WObj:=FakeWing;
        MoveL Target_1750,v30,fine,DrillTool\WObj:=FakeWing;
SetDO drillDone,1;
WaitUntil drillDone = 0;
        MoveL RelTool(Target_1750,0,0,-10),v30,z10,DrillTool\WObj:=FakeWing;
        MoveL RelTool(Target_1760,0,0,-10),v30,z10,DrillTool\WObj:=FakeWing;
        MoveL Target_1760,v30,fine,DrillTool\WObj:=FakeWing;
SetDO drillDone,1;
WaitUntil drillDone = 0;
        MoveL RelTool(Target_1760,0,0,-10),v30,z10,DrillTool\WObj:=FakeWing;
        MoveL RelTool(Target_1770,0,0,-10),v30,z10,DrillTool\WObj:=FakeWing;
        MoveL Target_1770,v30,fine,DrillTool\WObj:=FakeWing;
SetDO drillDone,1;
WaitUntil drillDone = 0;
        MoveL RelTool(Target_1770,0,0,-10),v30,z10,DrillTool\WObj:=FakeWing;
        MoveL RelTool(Target_1780,0,0,-10),v30,z10,DrillTool\WObj:=FakeWing;
        MoveL Target_1780,v30,fine,DrillTool\WObj:=FakeWing;
SetDO drillDone,1;
WaitUntil drillDone = 0;
        MoveL RelTool(Target_1780,0,0,-10),v30,z10,DrillTool\WObj:=FakeWing;
        MoveL RelTool(Target_1790,0,0,-10),v30,z10,DrillTool\WObj:=FakeWing;
        MoveL Target_1790,v30,fine,DrillTool\WObj:=FakeWing;
SetDO drillDone,1;
WaitUntil drillDone = 0;
        MoveL RelTool(Target_1790,0,0,-10),v30,z10,DrillTool\WObj:=FakeWing;
        MoveL RelTool(Target_1800,0,0,-10),v30,z10,DrillTool\WObj:=FakeWing;
        MoveL Target_1800,v30,fine,DrillTool\WObj:=FakeWing;
SetDO drillDone,1;
WaitUntil drillDone = 0;
        MoveL RelTool(Target_1800,0,0,-10),v30,z10,DrillTool\WObj:=FakeWing;
        MoveL RelTool(Target_1810,0,0,-10),v30,z10,DrillTool\WObj:=FakeWing;
        MoveL Target_1810,v30,fine,DrillTool\WObj:=FakeWing;
SetDO drillDone,1;
WaitUntil drillDone = 0;
        MoveL RelTool(Target_1810,0,0,-10),v30,z10,DrillTool\WObj:=FakeWing;
        MoveL RelTool(Target_1820,0,0,-10),v30,z10,DrillTool\WObj:=FakeWing;
        MoveL Target_1820,v30,fine,DrillTool\WObj:=FakeWing;
SetDO drillDone,1;
WaitUntil drillDone = 0;
        MoveL RelTool(Target_1820,0,0,-10),v30,z10,DrillTool\WObj:=FakeWing;
        MoveL RelTool(Target_1830,0,0,-10),v30,z10,DrillTool\WObj:=FakeWing;
        MoveL Target_1830,v30,fine,DrillTool\WObj:=FakeWing;
SetDO drillDone,1;
WaitUntil drillDone = 0;
        MoveL RelTool(Target_1830,0,0,-10),v30,z10,DrillTool\WObj:=FakeWing;
        MoveL RelTool(Target_1840,0,0,-10),v30,z10,DrillTool\WObj:=FakeWing;
        MoveL Target_1840,v30,fine,DrillTool\WObj:=FakeWing;
SetDO drillDone,1;
WaitUntil drillDone = 0;
        MoveL RelTool(Target_1840,0,0,-10),v30,z10,DrillTool\WObj:=FakeWing;
        MoveL RelTool(Target_1850,0,0,-10),v30,z10,DrillTool\WObj:=FakeWing;
        MoveL Target_1850,v30,fine,DrillTool\WObj:=FakeWing;
SetDO drillDone,1;
WaitUntil drillDone = 0;
        MoveL RelTool(Target_1850,0,0,-10),v30,z10,DrillTool\WObj:=FakeWing;
        MoveL RelTool(Target_1860,0,0,-10),v30,z10,DrillTool\WObj:=FakeWing;
        MoveL Target_1860,v30,fine,DrillTool\WObj:=FakeWing;
SetDO drillDone,1;
WaitUntil drillDone = 0;
        MoveL RelTool(Target_1860,0,0,-10),v30,z10,DrillTool\WObj:=FakeWing;
        MoveL RelTool(Target_1870,0,0,-10),v30,z10,DrillTool\WObj:=FakeWing;
        MoveL Target_1870,v30,fine,DrillTool\WObj:=FakeWing;
SetDO drillDone,1;
WaitUntil drillDone = 0;
        MoveL RelTool(Target_1870,0,0,-10),v30,z10,DrillTool\WObj:=FakeWing;
        MoveL RelTool(Target_1880,0,0,-10),v30,z10,DrillTool\WObj:=FakeWing;
        MoveL Target_1880,v30,fine,DrillTool\WObj:=FakeWing;
SetDO drillDone,1;
WaitUntil drillDone = 0;
        MoveL RelTool(Target_1880,0,0,-10),v30,z10,DrillTool\WObj:=FakeWing;
        MoveL RelTool(Target_1890,0,0,-10),v30,z10,DrillTool\WObj:=FakeWing;
        MoveL Target_1890,v30,fine,DrillTool\WObj:=FakeWing;
SetDO drillDone,1;
WaitUntil drillDone = 0;
        MoveL RelTool(Target_1890,0,0,-10),v30,z10,DrillTool\WObj:=FakeWing;
        MoveL RelTool(Target_1900,0,0,-10),v30,z10,DrillTool\WObj:=FakeWing;
        MoveL Target_1900,v30,fine,DrillTool\WObj:=FakeWing;
SetDO drillDone,1;
WaitUntil drillDone = 0;
        MoveL RelTool(Target_1900,0,0,-10),v30,z10,DrillTool\WObj:=FakeWing;
        MoveL RelTool(Target_1910,0,0,-10),v30,z10,DrillTool\WObj:=FakeWing;
        MoveL Target_1910,v30,fine,DrillTool\WObj:=FakeWing;
SetDO drillDone,1;
WaitUntil drillDone = 0;
        MoveL RelTool(Target_1910,0,0,-10),v30,z10,DrillTool\WObj:=FakeWing;
        MoveL RelTool(Target_1920,0,0,-10),v30,z10,DrillTool\WObj:=FakeWing;
        MoveL Target_1920,v30,fine,DrillTool\WObj:=FakeWing;
SetDO drillDone,1;
WaitUntil drillDone = 0;
        MoveL RelTool(Target_1920,0,0,-10),v30,z10,DrillTool\WObj:=FakeWing;
        MoveL RelTool(Target_1930,0,0,-10),v30,z10,DrillTool\WObj:=FakeWing;
        MoveL Target_1930,v30,fine,DrillTool\WObj:=FakeWing;
SetDO drillDone,1;
WaitUntil drillDone = 0;
        MoveL RelTool(Target_1930,0,0,-10),v30,z10,DrillTool\WObj:=FakeWing;
        MoveL RelTool(Target_1940,0,0,-10),v30,z10,DrillTool\WObj:=FakeWing;
        MoveL Target_1940,v30,fine,DrillTool\WObj:=FakeWing;
SetDO drillDone,1;
WaitUntil drillDone = 0;
        MoveL RelTool(Target_1940,0,0,-10),v30,z10,DrillTool\WObj:=FakeWing;
        MoveL RelTool(Target_1950,0,0,-10),v30,z10,DrillTool\WObj:=FakeWing;
        MoveL Target_1950,v30,fine,DrillTool\WObj:=FakeWing;
SetDO drillDone,1;
WaitUntil drillDone = 0;
        MoveL RelTool(Target_1950,0,0,-10),v30,z10,DrillTool\WObj:=FakeWing;
        MoveL RelTool(Target_1960,0,0,-10),v30,z10,DrillTool\WObj:=FakeWing;
        MoveL Target_1960,v30,fine,DrillTool\WObj:=FakeWing;
SetDO drillDone,1;
WaitUntil drillDone = 0;
        MoveL RelTool(Target_1960,0,0,-10),v30,z10,DrillTool\WObj:=FakeWing;
        MoveL RelTool(Target_1970,0,0,-10),v30,z10,DrillTool\WObj:=FakeWing;
        MoveL Target_1970,v30,fine,DrillTool\WObj:=FakeWing;
SetDO drillDone,1;
WaitUntil drillDone = 0;
        MoveL RelTool(Target_1970,0,0,-10),v30,z10,DrillTool\WObj:=FakeWing;
        MoveL RelTool(Target_1980,0,0,-10),v30,z10,DrillTool\WObj:=FakeWing;
        MoveL Target_1980,v30,fine,DrillTool\WObj:=FakeWing;
SetDO drillDone,1;
WaitUntil drillDone = 0;
        MoveL RelTool(Target_1980,0,0,-10),v30,z10,DrillTool\WObj:=FakeWing;
        MoveL RelTool(Target_1990,0,0,-10),v30,z10,DrillTool\WObj:=FakeWing;
        MoveL Target_1990,v30,fine,DrillTool\WObj:=FakeWing;
SetDO drillDone,1;
WaitUntil drillDone = 0;
        MoveL RelTool(Target_1990,0,0,-10),v30,z10,DrillTool\WObj:=FakeWing;
        MoveL RelTool(Target_2000,0,0,-10),v30,z10,DrillTool\WObj:=FakeWing;
        MoveL Target_2000,v30,fine,DrillTool\WObj:=FakeWing;
SetDO drillDone,1;
WaitUntil drillDone = 0;
        MoveL RelTool(Target_2000,0,0,-10),v30,z10,DrillTool\WObj:=FakeWing;
        MoveL RelTool(Target_2010,0,0,-10),v30,z10,DrillTool\WObj:=FakeWing;
        MoveL Target_2010,v30,fine,DrillTool\WObj:=FakeWing;
SetDO drillDone,1;
WaitUntil drillDone = 0;
        MoveL RelTool(Target_2010,0,0,-10),v30,z10,DrillTool\WObj:=FakeWing;
        MoveL RelTool(Target_2020,0,0,-10),v30,z10,DrillTool\WObj:=FakeWing;
        MoveL Target_2020,v30,fine,DrillTool\WObj:=FakeWing;
SetDO drillDone,1;
WaitUntil drillDone = 0;
        MoveL RelTool(Target_2020,0,0,-10),v30,z10,DrillTool\WObj:=FakeWing;
        MoveL RelTool(Target_2030,0,0,-10),v30,z10,DrillTool\WObj:=FakeWing;
        MoveL Target_2030,v30,fine,DrillTool\WObj:=FakeWing;
SetDO drillDone,1;
WaitUntil drillDone = 0;
        MoveL RelTool(Target_2030,0,0,-10),v30,z10,DrillTool\WObj:=FakeWing;
        MoveL RelTool(Target_2040,0,0,-10),v30,z10,DrillTool\WObj:=FakeWing;
        MoveL Target_2040,v30,fine,DrillTool\WObj:=FakeWing;
SetDO drillDone,1;
WaitUntil drillDone = 0;
        MoveL RelTool(Target_2040,0,0,-10),v30,z10,DrillTool\WObj:=FakeWing;
        MoveL RelTool(Target_2050,0,0,-10),v30,z10,DrillTool\WObj:=FakeWing;
        MoveL Target_2050,v30,fine,DrillTool\WObj:=FakeWing;
SetDO drillDone,1;
WaitUntil drillDone = 0;
        MoveL RelTool(Target_2050,0,0,-10),v30,z10,DrillTool\WObj:=FakeWing;
        MoveL RelTool(Target_2060,0,0,-10),v30,z10,DrillTool\WObj:=FakeWing;
        MoveL Target_2060,v30,fine,DrillTool\WObj:=FakeWing;
SetDO drillDone,1;
WaitUntil drillDone = 0;
        MoveL RelTool(Target_2060,0,0,-10),v30,z10,DrillTool\WObj:=FakeWing;
        MoveL RelTool(Target_2070,0,0,-10),v30,z10,DrillTool\WObj:=FakeWing;
        MoveL Target_2070,v30,fine,DrillTool\WObj:=FakeWing;
SetDO drillDone,1;
WaitUntil drillDone = 0;
        MoveL RelTool(Target_2070,0,0,-10),v30,z10,DrillTool\WObj:=FakeWing;
        MoveL RelTool(Target_2080,0,0,-10),v30,z10,DrillTool\WObj:=FakeWing;
        MoveL Target_2080,v30,fine,DrillTool\WObj:=FakeWing;
SetDO drillDone,1;
WaitUntil drillDone = 0;
        MoveL RelTool(Target_2080,0,0,-10),v30,z10,DrillTool\WObj:=FakeWing;
        MoveL RelTool(Target_2090,0,0,-10),v30,z10,DrillTool\WObj:=FakeWing;
        MoveL Target_2090,v30,fine,DrillTool\WObj:=FakeWing;
SetDO drillDone,1;
WaitUntil drillDone = 0;
        MoveL RelTool(Target_2090,0,0,-10),v30,z10,DrillTool\WObj:=FakeWing;
        MoveL RelTool(Target_2100,0,0,-10),v30,z10,DrillTool\WObj:=FakeWing;
        MoveL Target_2100,v30,fine,DrillTool\WObj:=FakeWing;
SetDO drillDone,1;
WaitUntil drillDone = 0;
        MoveL RelTool(Target_2100,0,0,-10),v30,z10,DrillTool\WObj:=FakeWing;
        MoveL RelTool(Target_2110,0,0,-10),v30,z10,DrillTool\WObj:=FakeWing;
        MoveL Target_2110,v30,fine,DrillTool\WObj:=FakeWing;
SetDO drillDone,1;
WaitUntil drillDone = 0;
        MoveL RelTool(Target_2110,0,0,-10),v30,z10,DrillTool\WObj:=FakeWing;
        MoveL RelTool(Target_2120,0,0,-10),v30,z10,DrillTool\WObj:=FakeWing;
        MoveL Target_2120,v30,fine,DrillTool\WObj:=FakeWing;
SetDO drillDone,1;
WaitUntil drillDone = 0;
        MoveL RelTool(Target_2120,0,0,-10),v30,z10,DrillTool\WObj:=FakeWing;
        MoveL RelTool(Target_2130,0,0,-10),v30,z10,DrillTool\WObj:=FakeWing;
        MoveL Target_2130,v30,fine,DrillTool\WObj:=FakeWing;
SetDO drillDone,1;
WaitUntil drillDone = 0;
        MoveL RelTool(Target_2130,0,0,-10),v30,z10,DrillTool\WObj:=FakeWing;
        MoveL RelTool(Target_2140,0,0,-10),v30,z10,DrillTool\WObj:=FakeWing;
        MoveL Target_2140,v30,fine,DrillTool\WObj:=FakeWing;
SetDO drillDone,1;
WaitUntil drillDone = 0;
        MoveL RelTool(Target_2140,0,0,-10),v30,z10,DrillTool\WObj:=FakeWing;
        MoveL RelTool(Target_2150,0,0,-10),v30,z10,DrillTool\WObj:=FakeWing;
        MoveL Target_2150,v30,fine,DrillTool\WObj:=FakeWing;
SetDO drillDone,1;
WaitUntil drillDone = 0;
        MoveL RelTool(Target_2150,0,0,-10),v30,z10,DrillTool\WObj:=FakeWing;
        MoveL RelTool(Target_2160,0,0,-10),v30,z10,DrillTool\WObj:=FakeWing;
        MoveL Target_2160,v30,fine,DrillTool\WObj:=FakeWing;
SetDO drillDone,1;
WaitUntil drillDone = 0;
        MoveL RelTool(Target_2160,0,0,-10),v30,z10,DrillTool\WObj:=FakeWing;
        MoveL RelTool(Target_2170,0,0,-10),v30,z10,DrillTool\WObj:=FakeWing;
        MoveL Target_2170,v30,fine,DrillTool\WObj:=FakeWing;
SetDO drillDone,1;
WaitUntil drillDone = 0;
        MoveL RelTool(Target_2170,0,0,-10),v30,z10,DrillTool\WObj:=FakeWing;
        MoveL RelTool(Target_2180,0,0,-10),v30,z10,DrillTool\WObj:=FakeWing;
        MoveL Target_2180,v30,fine,DrillTool\WObj:=FakeWing;
SetDO drillDone,1;
WaitUntil drillDone = 0;
        MoveL RelTool(Target_2180,0,0,-10),v30,z10,DrillTool\WObj:=FakeWing;
        MoveL RelTool(Target_2190,0,0,-10),v30,z10,DrillTool\WObj:=FakeWing;
        MoveL Target_2190,v30,fine,DrillTool\WObj:=FakeWing;
SetDO drillDone,1;
WaitUntil drillDone = 0;
        MoveL RelTool(Target_2190,0,0,-10),v30,z10,DrillTool\WObj:=FakeWing;
        MoveL RelTool(Target_2200,0,0,-10),v30,z10,DrillTool\WObj:=FakeWing;
        MoveL Target_2200,v30,fine,DrillTool\WObj:=FakeWing;
SetDO drillDone,1;
WaitUntil drillDone = 0;
        MoveL RelTool(Target_2200,0,0,-10),v30,z10,DrillTool\WObj:=FakeWing;
        MoveL RelTool(Target_2210,0,0,-10),v30,z10,DrillTool\WObj:=FakeWing;
        MoveL Target_2210,v30,fine,DrillTool\WObj:=FakeWing;
SetDO drillDone,1;
WaitUntil drillDone = 0;
        MoveL RelTool(Target_2210,0,0,-10),v30,z10,DrillTool\WObj:=FakeWing;
        MoveL RelTool(Target_2220,0,0,-10),v30,z10,DrillTool\WObj:=FakeWing;
        MoveL Target_2220,v30,fine,DrillTool\WObj:=FakeWing;
SetDO drillDone,1;
WaitUntil drillDone = 0;
